KUKA KRL program: EPS_2_26115_SA6998_A_20260219035530.src

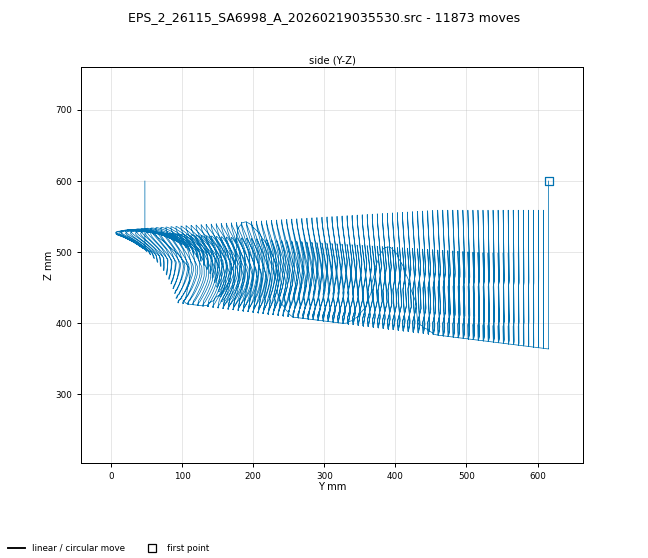
[picture p0: tool path of EPS_2_26115_SA6998_A_20260219035530.src, 11873 of 11875 moves have a stored position in this frame; points joined in program order, loops and branches not executed]
&ACCESS RVP
&REL 4
&COMMENT QRS 19112012
&PARAM EDITMASK = *
DEF PART()
EXT BAS (BAS_COMMAND :IN,REAL :IN )
INT I
BAS (#INITMOV,0 )

;KUKA QRS Post kuka4.cps  Date:22-06-2017 !

File_ID=3053

QRS_PRE_INIT()

;Init var - Until changes are made in qrs_pre_init
Outlet_Square_prg=0
Inlet_1_Square_prg=0
Inlet_2_Square_prg=0
Inlet_3_Square_prg=0
Inlet_4_Square_prg=0
Inlet_5_Square_prg=0

Outlet_1={X 0.000, Y 460.000, Z 458.500, B 0.000, E1 0.000 }
Inlet_1={X 0.000, Y 525.210, Z 398.500, B 0.000, E1 203.000 }
Outlet_1_type=201
Inlet_1_type=201
;QRS#1=Sidecore dimensions
;QRS#2=200-8" PVC SDR 35 Cut Back
;QRS#3=200-8" PVC SDR 35
;QRS#4=
;QRS#5=
;QRS#6=
;QRS#7=
;QRS#8=
;QRS#9=12-08 PSX
;QRS#10=12-08 PSX
;QRS#11=
;QRS#12=
;QRS#13=
;QRS#14=
;QRS#15=
;QRS#16=1220x127x838 2,75'
;QRS#17=EPS Height
;QRS#18=559
;QRS#19=*
;QRS#20= UPDATED VERSION 22-06-2017
;QRS#21=*
Outlet_Square=0100
Inlet_1_Square=0100
Inlet_2_Square=0
Inlet_3_Square=0
Inlet_4_Square=0
Inlet_5_Square=0
Mill_Square=1
Outlet_Square_Prg=214
Inlet_1_Square_prg=204

QRS_INIT()

$ADVANCE=5

; T1
PTP {E1 173.606,E2 173.606}
PTP {X 0,Y 615.505,A -85,B 0,C 180,E1 173.606,E2 173.606,E3 0,E4 0,E5 0,E6 0}
QRS_SPEED_INIT()
LIN {X 0,Y 615.505,Z 600,A -85,B 0,C 180,E1 173.606,E2 173.606,E3 0,E4 0,E5 0,E6 0} C_VEL
LIN {X 0,Y 615.505,Z 373.876,A -85,B 0,C 180,E1 173.606,E2 173.606} C_VEL
LIN {X 0,Y 615.505,Z 365.698,A -85,B 0,C 180,E1 173.606,E2 173.606} C_VEL
LIN {X 0,Y 615.491,Z 363.698,A -85,B 0,C 180,E1 173.42,E2 173.42} C_VEL
LIN {X 0,Y 615.494,Z 363.698,A -85,B 0,C 180,E1 170.801,E2 170.801} C_VEL
LIN {X 0,Y 615.477,Z 363.7,A -85,B 0,C 180,E1 168.139,E2 168.139} C_VEL
LIN {X 0,Y 615.491,Z 363.701,A -85,B 0,C 180,E1 165.451,E2 165.451} C_VEL
LIN {X 0,Y 615.482,Z 363.699,A -85,B 0,C 180,E1 162.729,E2 162.729} C_VEL
LIN {X 0,Y 615.481,Z 363.7,A -85,B 0,C 180,E1 159.967,E2 159.967} C_VEL
LIN {X 0,Y 615.493,Z 363.701,A -85,B 0,C 180,E1 157.156,E2 157.156} C_VEL
LIN {X 0,Y 615.477,Z 363.701,A -85,B 0,C 180,E1 154.284,E2 154.284} C_VEL
LIN {X 0,Y 615.487,Z 363.698,A -85,B 0,C 180,E1 151.55,E2 151.55} C_VEL
LIN {X 0,Y 615.492,Z 363.7,A -85,B 0,C 180,E1 148.914,E2 148.914} C_VEL
LIN {X 0,Y 615.48,Z 363.7,A -85,B 0,C 180,E1 146.467,E2 146.467} C_VEL
LIN {X 0,Y 615.492,Z 363.7,A -85,B 0,C 180,E1 143.575,E2 143.575} C_VEL
LIN {X 0,Y 615.482,Z 363.699,A -85,B 0,C 180,E1 140.939,E2 140.939} C_VEL
LIN {X 0,Y 615.491,Z 363.701,A -85,B 0,C 180,E1 138.526,E2 138.526} C_VEL
LIN {X 0,Y 615.48,Z 363.699,A -85,B 0,C 180,E1 135.85,E2 135.85} C_VEL
LIN {X 0,Y 615.482,Z 363.7,A -85,B 0,C 180,E1 133.047,E2 133.047} C_VEL
LIN {X 0,Y 615.472,Z 363.701,A -85,B 0,C 180,E1 130.608,E2 130.608} C_VEL
LIN {X 0,Y 615.489,Z 363.701,A -85,B 0,C 180,E1 128.012,E2 128.012} C_VEL
LIN {X 0,Y 615.498,Z 363.695,A -85,B 0,C 180,E1 125.616,E2 125.616} C_VEL
LIN {X 0,Y 615.489,Z 363.698,A -85,B 0,C 180,E1 123.237,E2 123.237} C_VEL
LIN {X 0,Y 615.496,Z 363.7,A -85,B 0,C 180,E1 120.92,E2 120.92} C_VEL
LIN {X 0,Y 615.478,Z 363.7,A -85,B 0,C 180,E1 118.448,E2 118.448} C_VEL
LIN {X 0,Y 615.486,Z 363.701,A -85,B 0,C 180,E1 115.568,E2 115.568} C_VEL
LIN {X 0,Y 615.48,Z 363.7,A -85,B 0,C 180,E1 112.846,E2 112.846} C_VEL
LIN {X 0,Y 615.489,Z 363.697,A -85,B 0,C 180,E1 110.034,E2 110.034} C_VEL
LIN {X 0,Y 615.491,Z 363.7,A -85,B 0,C 180,E1 107.271,E2 107.271} C_VEL
LIN {X 0,Y 615.481,Z 363.7,A -85,B 0,C 180,E1 104.55,E2 104.55} C_VEL
LIN {X 0,Y 615.478,Z 363.7,A -85,B 0,C 180,E1 102.531,E2 102.531} C_VEL
LIN {X 0,Y 615.489,Z 365.87,A -85,B 0,C 180,E1 100.528,E2 100.528} C_VEL
LIN {X 0,Y 615.493,Z 369.04,A -85,B 0,C 180,E1 97.877,E2 97.877} C_VEL
LIN {X 0,Y 615.456,Z 372.376,A -85,B 0,C 180,E1 95.243,E2 95.243} C_VEL
LIN {X 0,Y 615.448,Z 374.929,A -85,B 0,C 180,E1 93.274,E2 93.274} C_VEL
LIN {X 0,Y 615.441,Z 377.52,A -85,B 0,C 180,E1 91.31,E2 91.31} C_VEL
LIN {X 0,Y 615.434,Z 380.15,A -85,B 0,C 180,E1 89.347,E2 89.347} C_VEL
LIN {X 0,Y 615.428,Z 382.818,A -85,B 0,C 180,E1 87.383,E2 87.383} C_VEL
LIN {X 0,Y 615.426,Z 385.523,A -85,B 0,C 180,E1 85.416,E2 85.416} C_VEL
LIN {X 0,Y 615.431,Z 388.264,A -85,B 0,C 180,E1 83.444,E2 83.444} C_VEL
LIN {X 0,Y 615.434,Z 391.045,A -85,B 0,C 180,E1 81.464,E2 81.464} C_VEL
LIN {X 0,Y 615.435,Z 394.349,A -85,B 0,C 180,E1 79.138,E2 79.138} C_VEL
LIN {X 0,Y 615.478,Z 395.234,A -85,B 0,C 180,E1 78.537,E2 78.537} C_VEL
LIN {X 0,Y 615.495,Z 407.591,A -85,B 0,C 180,E1 78.266,E2 78.266} C_VEL
LIN {X 0,Y 615.465,Z 420.48,A -85,B 0,C 180,E1 77.848,E2 77.848} C_VEL
LIN {X 0,Y 615.439,Z 432.744,A -85,B 0,C 180,E1 77.303,E2 77.303} C_VEL
LIN {X 0,Y 615.477,Z 444.293,A -85,B 0,C 180,E1 76.632,E2 76.632} C_VEL
LIN {X 0,Y 615.498,Z 454.263,A -85,B 0,C 180,E1 75.911,E2 75.911} C_VEL
LIN {X 0,Y 615.497,Z 463.3,A -85,B 0,C 180,E1 75.115,E2 75.115} C_VEL
LIN {X 0,Y 615.496,Z 472.571,A -85,B 0,C 180,E1 74.097,E2 74.097} C_VEL
LIN {X 0,Y 615.497,Z 480.051,A -85,B 0,C 180,E1 73.074,E2 73.074} C_VEL
LIN {X 0,Y 615.497,Z 486.008,A -85,B 0,C 180,E1 72.045,E2 72.045} C_VEL
LIN {X 0,Y 615.496,Z 490.667,A -85,B 0,C 180,E1 71.01,E2 71.01} C_VEL
LIN {X 0,Y 615.498,Z 494.172,A -85,B 0,C 180,E1 69.969,E2 69.969} C_VEL
LIN {X 0,Y 615.492,Z 495.899,A -85,B 0,C 180,E1 69.271,E2 69.271} C_VEL
LIN {X 0,Y 615.497,Z 497.187,A -85,B 0,C 180,E1 68.57,E2 68.57} C_VEL
LIN {X 0,Y 615.491,Z 498.143,A -85,B 0,C 180,E1 67.654,E2 67.654} C_VEL
LIN {X 0,Y 615.496,Z 498.27,A -85,B 0,C 180,E1 66.446,E2 66.446} C_VEL
LIN {X 0,Y 615.494,Z 497.679,A -85,B 0,C 180,E1 65.73,E2 65.73} C_VEL
LIN {X 0,Y 615.495,Z 495.447,A -85,B 0,C 180,E1 64.43,E2 64.43} C_VEL
LIN {X 0,Y 615.498,Z 492.002,A -85,B 0,C 180,E1 63.257,E2 63.257} C_VEL
LIN {X 0,Y 615.495,Z 487.093,A -85,B 0,C 180,E1 62.087,E2 62.087} C_VEL
LIN {X 0,Y 615.496,Z 480.902,A -85,B 0,C 180,E1 60.971,E2 60.971} C_VEL
LIN {X 0,Y 615.497,Z 474.27,A -85,B 0,C 180,E1 60.023,E2 60.023} C_VEL
LIN {X 0,Y 615.497,Z 466.126,A -85,B 0,C 180,E1 59.083,E2 59.083} C_VEL
LIN {X 0,Y 615.499,Z 456.191,A -85,B 0,C 180,E1 58.156,E2 58.156} C_VEL
LIN {X 0,Y 615.496,Z 446.877,A -85,B 0,C 180,E1 57.448,E2 57.448} C_VEL
LIN {X 0,Y 615.477,Z 435.697,A -85,B 0,C 180,E1 56.765,E2 56.765} C_VEL
LIN {X 0,Y 615.487,Z 422.997,A -85,B 0,C 180,E1 56.163,E2 56.163} C_VEL
LIN {X 0,Y 615.486,Z 410.581,A -85,B 0,C 180,E1 55.726,E2 55.726} C_VEL
LIN {X 0,Y 615.492,Z 397.092,A -85,B 0,C 180,E1 55.407,E2 55.407} C_VEL
LIN {X 0,Y 615.489,Z 395.187,A -85,B 0,C 180,E1 55.364,E2 55.364} C_VEL
LIN {X 0,Y 615.474,Z 391.482,A -85,B 0,C 180,E1 52.759,E2 52.759} C_VEL
LIN {X 0,Y 615.493,Z 387.48,A -85,B 0,C 180,E1 49.911,E2 49.911} C_VEL
LIN {X 0,Y 615.479,Z 384.358,A -85,B 0,C 180,E1 47.649,E2 47.649} C_VEL
LIN {X 0,Y 615.46,Z 380.643,A -85,B 0,C 180,E1 44.932,E2 44.932} C_VEL
LIN {X 0,Y 615.495,Z 376.831,A -85,B 0,C 180,E1 42.084,E2 42.084} C_VEL
LIN {X 0,Y 615.45,Z 373.787,A -85,B 0,C 180,E1 39.753,E2 39.753} C_VEL
LIN {X 0,Y 615.457,Z 370.168,A -85,B 0,C 180,E1 36.936,E2 36.936} C_VEL
LIN {X 0,Y 615.495,Z 366.665,A -85,B 0,C 180,E1 34.022,E2 34.022} C_VEL
LIN {X 0,Y 615.485,Z 363.854,A -85,B 0,C 180,E1 31.686,E2 31.686} C_VEL
LIN {X 0,Y 615.463,Z 363.7,A -85,B 0,C 180,E1 29.408,E2 29.408} C_VEL
LIN {X 0,Y 615.481,Z 363.695,A -85,B 0,C 180,E1 27.049,E2 27.049} C_VEL
LIN {X 0,Y 615.471,Z 363.697,A -85,B 0,C 180,E1 24.273,E2 24.273} C_VEL
LIN {X 0,Y 615.486,Z 363.701,A -85,B 0,C 180,E1 22.137,E2 22.137} C_VEL
LIN {X 0,Y 615.491,Z 363.698,A -85,B 0,C 180,E1 19.338,E2 19.338} C_VEL
LIN {X 0,Y 615.466,Z 363.7,A -85,B 0,C 180,E1 16.432,E2 16.432} C_VEL
LIN {X 0,Y 615.478,Z 363.7,A -85,B 0,C 180,E1 13.874,E2 13.874} C_VEL
LIN {X 0,Y 615.489,Z 363.693,A -85,B 0,C 180,E1 10.902,E2 10.902} C_VEL
LIN {X 0,Y 615.482,Z 363.7,A -85,B 0,C 180,E1 8.537,E2 8.537} C_VEL
LIN {X 0,Y 615.49,Z 363.7,A -85,B 0,C 180,E1 5.898,E2 5.898} C_VEL
LIN {X 0,Y 615.49,Z 363.702,A -85,B 0,C 180,E1 3.273,E2 3.273} C_VEL
LIN {X 0,Y 615.491,Z 363.7,A -85,B 0,C 180,E1 0.654,E2 0.654} C_VEL
LIN {X 0,Y 615.486,Z 363.699,A -85,B 0,C 180,E1 -1.963,E2 -1.963} C_VEL
LIN {X 0,Y 615.476,Z 363.7,A -85,B 0,C 180,E1 -4.585,E2 -4.585} C_VEL
LIN {X 0,Y 615.492,Z 363.695,A -85,B 0,C 180,E1 -7.216,E2 -7.216} C_VEL
LIN {X 0,Y 615.468,Z 363.7,A -85,B 0,C 180,E1 -9.863,E2 -9.863} C_VEL
LIN {X 0,Y 615.468,Z 363.699,A -85,B 0,C 180,E1 -12.531,E2 -12.531} C_VEL
LIN {X 0,Y 615.483,Z 363.696,A -85,B 0,C 180,E1 -15.226,E2 -15.226} C_VEL
LIN {X 0,Y 615.465,Z 363.7,A -85,B 0,C 180,E1 -17.958,E2 -17.958} C_VEL
LIN {X 0,Y 615.493,Z 363.695,A -85,B 0,C 180,E1 -20.731,E2 -20.731} C_VEL
LIN {X 0,Y 615.486,Z 363.699,A -85,B 0,C 180,E1 -23.557,E2 -23.557} C_VEL
LIN {X 0,Y 615.458,Z 363.7,A -85,B 0,C 180,E1 -25.717,E2 -25.717} C_VEL
LIN {X 0,Y 615.481,Z 363.695,A -85,B 0,C 180,E1 -28.454,E2 -28.454} C_VEL
LIN {X 0,Y 615.469,Z 363.698,A -85,B 0,C 180,E1 -31.088,E2 -31.088} C_VEL
LIN {X 0,Y 615.468,Z 363.7,A -85,B 0,C 180,E1 -33.535,E2 -33.535} C_VEL
LIN {X 0,Y 615.491,Z 363.7,A -85,B 0,C 180,E1 -35.838,E2 -35.838} C_VEL
LIN {X 0,Y 615.463,Z 363.699,A -85,B 0,C 180,E1 -38.071,E2 -38.071} C_VEL
LIN {X 0,Y 615.492,Z 363.692,A -85,B 0,C 180,E1 -40.606,E2 -40.606} C_VEL
LIN {X 0,Y 615.459,Z 363.7,A -85,B 0,C 180,E1 -43.247,E2 -43.247} C_VEL
LIN {X 0,Y 615.472,Z 363.697,A -85,B 0,C 180,E1 -46.004,E2 -46.004} C_VEL
LIN {X 0,Y 615.475,Z 363.696,A -85,B 0,C 180,E1 -48.907,E2 -48.907} C_VEL
LIN {X 0,Y 615.47,Z 363.7,A -85,B 0,C 180,E1 -51.097,E2 -51.097} C_VEL
LIN {X 0,Y 615.483,Z 363.702,A -85,B 0,C 180,E1 -53.577,E2 -53.577} C_VEL
LIN {X 0,Y 615.493,Z 363.825,A -85,B 0,C 180,E1 -54.538,E2 -54.538} C_VEL
LIN {X 0,Y 615.444,Z 372.587,A -85,B 0,C 180,E1 -57.154,E2 -57.154} C_VEL
LIN {X 0,Y 615.423,Z 380.521,A -85,B 0,C 180,E1 -59.459,E2 -59.459} C_VEL
LIN {X 0,Y 615.479,Z 389.763,A -85,B 0,C 180,E1 -62.087,E2 -62.087} C_VEL
LIN {X 0,Y 615.455,Z 399.275,A -85,B 0,C 180,E1 -64.721,E2 -64.721} C_VEL
LIN {X 0,Y 615.46,Z 408.245,A -85,B 0,C 180,E1 -67.156,E2 -67.156} C_VEL
LIN {X 0,Y 615.489,Z 416.801,A -85,B 0,C 180,E1 -69.443,E2 -69.443} C_VEL
LIN {X 0,Y 615.486,Z 428.021,A -85,B 0,C 180,E1 -72.388,E2 -72.388} C_VEL
LIN {X 0,Y 615.482,Z 438.548,A -85,B 0,C 180,E1 -75.114,E2 -75.114} C_VEL
LIN {X 0,Y 615.469,Z 449.091,A -85,B 0,C 180,E1 -77.806,E2 -77.806} C_VEL
LIN {X 0,Y 615.494,Z 451.215,A -85,B 0,C 180,E1 -78.35,E2 -78.35} C_VEL
LIN {X 0,Y 615.497,Z 465.878,A -85,B 0,C 180,E1 -78.642,E2 -78.642} C_VEL
LIN {X 0,Y 615.457,Z 478.927,A -85,B 0,C 180,E1 -79.049,E2 -79.049} C_VEL
LIN {X 0,Y 615.452,Z 490.803,A -85,B 0,C 180,E1 -79.557,E2 -79.557} C_VEL
LIN {X 0,Y 615.496,Z 501.412,A -85,B 0,C 180,E1 -80.139,E2 -80.139} C_VEL
LIN {X 0,Y 615.498,Z 512.25,A -85,B 0,C 180,E1 -80.886,E2 -80.886} C_VEL
LIN {X 0,Y 615.497,Z 522.827,A -85,B 0,C 180,E1 -81.796,E2 -81.796} C_VEL
LIN {X 0,Y 615.497,Z 531.977,A -85,B 0,C 180,E1 -82.786,E2 -82.786} C_VEL
LIN {X 0,Y 615.497,Z 539.325,A -85,B 0,C 180,E1 -83.774,E2 -83.774} C_VEL
LIN {X 0,Y 615.498,Z 545.212,A -85,B 0,C 180,E1 -84.76,E2 -84.76} C_VEL
LIN {X 0,Y 615.494,Z 549.857,A -85,B 0,C 180,E1 -85.745,E2 -85.745} C_VEL
LIN {X 0,Y 615.494,Z 553.403,A -85,B 0,C 180,E1 -86.728,E2 -86.728} C_VEL
LIN {X 0,Y 615.497,Z 555.236,A -85,B 0,C 180,E1 -87.383,E2 -87.383} C_VEL
LIN {X 0,Y 615.499,Z 556.61,A -85,B 0,C 180,E1 -88.038,E2 -88.038} C_VEL
LIN {X 0,Y 615.496,Z 558.174,A -85,B 0,C 180,E1 -89.347,E2 -89.347} C_VEL
LIN {X 0,Y 615.494,Z 558.389,A -85,B 0,C 180,E1 -90.001,E2 -90.001} C_VEL
LIN {X 0,Y 615.495,Z 557.579,A -85,B 0,C 180,E1 -91.31,E2 -91.31} C_VEL
LIN {X 0,Y 615.499,Z 556.606,A -85,B 0,C 180,E1 -91.964,E2 -91.964} C_VEL
LIN {X 0,Y 615.497,Z 555.23,A -85,B 0,C 180,E1 -92.619,E2 -92.619} C_VEL
LIN {X 0,Y 615.496,Z 552.345,A -85,B 0,C 180,E1 -93.602,E2 -93.602} C_VEL
LIN {X 0,Y 615.498,Z 548.436,A -85,B 0,C 180,E1 -94.586,E2 -94.586} C_VEL
LIN {X 0,Y 615.499,Z 543.398,A -85,B 0,C 180,E1 -95.571,E2 -95.571} C_VEL
LIN {X 0,Y 615.497,Z 536.87,A -85,B 0,C 180,E1 -96.583,E2 -96.583} C_VEL
LIN {X 0,Y 615.497,Z 529.123,A -85,B 0,C 180,E1 -97.547,E2 -97.547} C_VEL
LIN {X 0,Y 615.498,Z 521.033,A -85,B 0,C 180,E1 -98.372,E2 -98.372} C_VEL
LIN {X 0,Y 615.499,Z 511.153,A -85,B 0,C 180,E1 -99.2,E2 -99.2} C_VEL
LIN {X 0,Y 615.487,Z 499.963,A -85,B 0,C 180,E1 -99.946,E2 -99.946} C_VEL
LIN {X 0,Y 615.449,Z 489.006,A -85,B 0,C 180,E1 -100.529,E2 -100.529} C_VEL
LIN {X 0,Y 615.463,Z 476.725,A -85,B 0,C 180,E1 -101.032,E2 -101.032} C_VEL
LIN {X 0,Y 615.499,Z 464.017,A -85,B 0,C 180,E1 -101.402,E2 -101.402} C_VEL
LIN {X 0,Y 615.495,Z 451.205,A -85,B 0,C 180,E1 -101.653,E2 -101.653} C_VEL
LIN {X 0,Y 615.471,Z 441.065,A -85,B 0,C 180,E1 -104.242,E2 -104.242} C_VEL
LIN {X 0,Y 615.49,Z 430.636,A -85,B 0,C 180,E1 -106.929,E2 -106.929} C_VEL
LIN {X 0,Y 615.484,Z 420.1,A -85,B 0,C 180,E1 -109.686,E2 -109.686} C_VEL
LIN {X 0,Y 615.491,Z 410.087,A -85,B 0,C 180,E1 -112.346,E2 -112.346} C_VEL
LIN {X 0,Y 615.445,Z 400.321,A -85,B 0,C 180,E1 -114.994,E2 -114.994} C_VEL
LIN {X 0,Y 615.476,Z 391.073,A -85,B 0,C 180,E1 -117.547,E2 -117.547} C_VEL
LIN {X 0,Y 615.439,Z 381.831,A -85,B 0,C 180,E1 -120.163,E2 -120.163} C_VEL
LIN {X 0,Y 615.433,Z 373.9,A -85,B 0,C 180,E1 -122.461,E2 -122.461} C_VEL
LIN {X 0,Y 615.46,Z 365.964,A -85,B 0,C 180,E1 -124.818,E2 -124.818} C_VEL
LIN {X 0,Y 615.495,Z 363.696,A -85,B 0,C 180,E1 -125.516,E2 -125.516} C_VEL
LIN {X 0,Y 615.491,Z 363.699,A -85,B 0,C 180,E1 -128.069,E2 -128.069} C_VEL
LIN {X 0,Y 615.481,Z 363.7,A -85,B 0,C 180,E1 -130.608,E2 -130.608} C_VEL
LIN {X 0,Y 615.484,Z 363.7,A -85,B 0,C 180,E1 -133.246,E2 -133.246} C_VEL
LIN {X 0,Y 615.473,Z 363.701,A -85,B 0,C 180,E1 -136.005,E2 -136.005} C_VEL
LIN {X 0,Y 615.491,Z 363.7,A -85,B 0,C 180,E1 -138.526,E2 -138.526} C_VEL
LIN {X 0,Y 615.484,Z 363.698,A -85,B 0,C 180,E1 -141.095,E2 -141.095} C_VEL
LIN {X 0,Y 615.494,Z 363.697,A -85,B 0,C 180,E1 -143.576,E2 -143.576} C_VEL
LIN {X 0,Y 615.492,Z 363.7,A -85,B 0,C 180,E1 -145.978,E2 -145.978} C_VEL
LIN {X 0,Y 615.477,Z 363.7,A -85,B 0,C 180,E1 -148.314,E2 -148.314} C_VEL
LIN {X 0,Y 615.475,Z 363.7,A -85,B 0,C 180,E1 -150.593,E2 -150.593} C_VEL
LIN {X 0,Y 615.486,Z 363.7,A -85,B 0,C 180,E1 -152.956,E2 -152.956} C_VEL
LIN {X 0,Y 615.476,Z 363.7,A -85,B 0,C 180,E1 -155.727,E2 -155.727} C_VEL
LIN {X 0,Y 615.474,Z 363.7,A -85,B 0,C 180,E1 -157.863,E2 -157.863} C_VEL
LIN {X 0,Y 615.486,Z 363.699,A -85,B 0,C 180,E1 -160.662,E2 -160.662} C_VEL
LIN {X 0,Y 615.488,Z 363.701,A -85,B 0,C 180,E1 -163.569,E2 -163.569} C_VEL
LIN {X 0,Y 615.473,Z 363.7,A -85,B 0,C 180,E1 -166.125,E2 -166.125} C_VEL
LIN {X 0,Y 615.495,Z 363.699,A -85,B 0,C 180,E1 -168.807,E2 -168.807} C_VEL
LIN {X 0,Y 615.488,Z 363.698,A -85,B 0,C 180,E1 -171.463,E2 -171.463} C_VEL
LIN {X 0,Y 615.482,Z 363.7,A -85,B 0,C 180,E1 -174.101,E2 -174.101} C_VEL
LIN {X 0,Y 615.482,Z 363.7,A -85,B 0,C 180,E1 -176.727,E2 -176.727} C_VEL
LIN {X 0,Y 615.479,Z 363.7,A -85,B 0,C 180,E1 -179.346,E2 -179.346} C_VEL
LIN {X 0,Y 615.485,Z 363.7,A -85,B 0,C 180,E1 -181.963,E2 -181.963} C_VEL
LIN {X 0,Y 615.488,Z 363.698,A -85,B 0,C 180,E1 -184.585,E2 -184.585} C_VEL
LIN {X 0,Y 615.491,Z 363.698,A -85,B 0,C 180,E1 -186.58,E2 -186.58} C_VEL
LIN {X 0,Y 614.818,Z 363.846,A -85,B 0,C 180,E1 -187.126,E2 -187.126} C_VEL
LIN {X 0,Y 611.987,Z 364.255,A -85,B 0,C 180,E1 -188.012,E2 -188.012} C_VEL
LIN {X 0,Y 609.594,Z 364.567,A -85,B 0,C 180,E1 -188.724,E2 -188.724} C_VEL
LIN {X 0,Y 608.554,Z 364.686,A -85,B 0,C 180,E1 -189.274,E2 -189.274} C_VEL
LIN {X 0,Y 608.461,Z 364.695,A -85,B 0,C 180,E1 -189.46,E2 -189.46} C_VEL
LIN {X 0,Y 608.457,Z 364.695,A -85,B 0,C 180,E1 -192,E2 -192} C_VEL
LIN {X 0,Y 608.478,Z 364.694,A -85,B 0,C 180,E1 -194.72,E2 -194.72} C_VEL
LIN {X 0,Y 608.449,Z 364.697,A -85,B 0,C 180,E1 -197.477,E2 -197.477} C_VEL
LIN {X 0,Y 608.459,Z 364.695,A -85,B 0,C 180,E1 -200.274,E2 -200.274} C_VEL
LIN {X 0,Y 608.452,Z 364.696,A -85,B 0,C 180,E1 -203.124,E2 -203.124} C_VEL
LIN {X 0,Y 608.464,Z 364.695,A -85,B 0,C 180,E1 -205.719,E2 -205.719} C_VEL
LIN {X 0,Y 608.451,Z 364.697,A -85,B 0,C 180,E1 -208.267,E2 -208.267} C_VEL
LIN {X 0,Y 608.479,Z 364.692,A -85,B 0,C 180,E1 -210.544,E2 -210.544} C_VEL
LIN {X 0,Y 608.463,Z 364.694,A -85,B 0,C 180,E1 -212.879,E2 -212.879} C_VEL
LIN {X 0,Y 608.441,Z 364.699,A -85,B 0,C 180,E1 -215.278,E2 -215.278} C_VEL
LIN {X 0,Y 608.464,Z 364.694,A -85,B 0,C 180,E1 -217.747,E2 -217.747} C_VEL
LIN {X 0,Y 608.448,Z 364.697,A -85,B 0,C 180,E1 -220.328,E2 -220.328} C_VEL
LIN {X 0,Y 608.467,Z 364.694,A -85,B 0,C 180,E1 -223.308,E2 -223.308} C_VEL
LIN {X 0,Y 608.472,Z 364.693,A -85,B 0,C 180,E1 -226.13,E2 -226.13} C_VEL
LIN {X 0,Y 608.456,Z 364.698,A -85,B 0,C 180,E1 -228.823,E2 -228.823} C_VEL
LIN {X 0,Y 608.441,Z 364.697,A -85,B 0,C 180,E1 -231.409,E2 -231.409} C_VEL
LIN {X 0,Y 608.453,Z 364.698,A -85,B 0,C 180,E1 -233.954,E2 -233.954} C_VEL
LIN {X 0,Y 608.47,Z 364.694,A -85,B 0,C 180,E1 -236.329,E2 -236.329} C_VEL
LIN {X 0,Y 608.466,Z 364.694,A -85,B 0,C 180,E1 -238.73,E2 -238.73} C_VEL
LIN {X 0,Y 608.473,Z 364.694,A -85,B 0,C 180,E1 -241.38,E2 -241.38} C_VEL
LIN {X 0,Y 608.479,Z 364.695,A -85,B 0,C 180,E1 -244.278,E2 -244.278} C_VEL
LIN {X 0,Y 608.45,Z 364.696,A -85,B 0,C 180,E1 -246.875,E2 -246.875} C_VEL
LIN {X 0,Y 608.47,Z 364.694,A -85,B 0,C 180,E1 -249.321,E2 -249.321} C_VEL
LIN {X 0,Y 608.453,Z 364.696,A -85,B 0,C 180,E1 -251.827,E2 -251.827} C_VEL
LIN {X 0,Y 608.474,Z 364.695,A -85,B 0,C 180,E1 -254.593,E2 -254.593} C_VEL
LIN {X 0,Y 608.473,Z 364.693,A -85,B 0,C 180,E1 -257.322,E2 -257.322} C_VEL
LIN {X 0,Y 608.428,Z 364.939,A -85,B 0,C 180,E1 -257.998,E2 -257.998} C_VEL
LIN {X 0,Y 608.435,Z 368.164,A -85,B 0,C 180,E1 -260.693,E2 -260.693} C_VEL
LIN {X 0,Y 608.418,Z 370.547,A -85,B 0,C 180,E1 -262.699,E2 -262.699} C_VEL
LIN {X 0,Y 608.392,Z 373.926,A -85,B 0,C 180,E1 -265.361,E2 -265.361} C_VEL
LIN {X 0,Y 608.464,Z 377.372,A -85,B 0,C 180,E1 -268.013,E2 -268.013} C_VEL
LIN {X 0,Y 608.382,Z 380.897,A -85,B 0,C 180,E1 -270.661,E2 -270.661} C_VEL
LIN {X 0,Y 608.362,Z 383.583,A -85,B 0,C 180,E1 -272.647,E2 -272.647} C_VEL
LIN {X 0,Y 608.362,Z 386.308,A -85,B 0,C 180,E1 -274.637,E2 -274.637} C_VEL
LIN {X 0,Y 608.385,Z 389.071,A -85,B 0,C 180,E1 -276.632,E2 -276.632} C_VEL
LIN {X 0,Y 608.38,Z 392.82,A -85,B 0,C 180,E1 -279.306,E2 -279.306} C_VEL
LIN {X 0,Y 608.407,Z 395.677,A -85,B 0,C 180,E1 -281.324,E2 -281.324} C_VEL
LIN {X 0,Y 608.544,Z 409.709,A -85,B 0,C 180,E1 -281.659,E2 -281.659} C_VEL
LIN {X 0,Y 608.495,Z 422.071,A -85,B 0,C 180,E1 -282.082,E2 -282.082} C_VEL
LIN {X 0,Y 608.459,Z 433.153,A -85,B 0,C 180,E1 -282.591,E2 -282.591} C_VEL
LIN {X 0,Y 608.475,Z 444.709,A -85,B 0,C 180,E1 -283.27,E2 -283.27} C_VEL
LIN {X 0,Y 608.472,Z 455.165,A -85,B 0,C 180,E1 -284.036,E2 -284.036} C_VEL
LIN {X 0,Y 608.468,Z 464.586,A -85,B 0,C 180,E1 -284.89,E2 -284.89} C_VEL
LIN {X 0,Y 608.461,Z 473.753,A -85,B 0,C 180,E1 -285.92,E2 -285.92} C_VEL
LIN {X 0,Y 608.46,Z 481.119,A -85,B 0,C 180,E1 -286.955,E2 -286.955} C_VEL
LIN {X 0,Y 608.455,Z 486.111,A -85,B 0,C 180,E1 -287.822,E2 -287.822} C_VEL
LIN {X 0,Y 608.456,Z 490.913,A -85,B 0,C 180,E1 -288.868,E2 -288.868} C_VEL
LIN {X 0,Y 608.436,Z 494.538,A -85,B 0,C 180,E1 -289.921,E2 -289.921} C_VEL
LIN {X 0,Y 608.423,Z 497.07,A -85,B 0,C 180,E1 -290.981,E2 -290.981} C_VEL
LIN {X 0,Y 608.417,Z 498.149,A -85,B 0,C 180,E1 -291.692,E2 -291.692} C_VEL
LIN {X 0,Y 608.423,Z 498.843,A -85,B 0,C 180,E1 -292.468,E2 -292.468} C_VEL
LIN {X 0,Y 608.432,Z 498.988,A -85,B 0,C 180,E1 -293.123,E2 -293.123} C_VEL
LIN {X 0,Y 608.422,Z 498.452,A -85,B 0,C 180,E1 -294.14,E2 -294.14} C_VEL
LIN {X 0,Y 608.439,Z 496.675,A -85,B 0,C 180,E1 -295.3,E2 -295.3} C_VEL
LIN {X 0,Y 608.432,Z 493.806,A -85,B 0,C 180,E1 -296.403,E2 -296.403} C_VEL
LIN {X 0,Y 608.436,Z 489.661,A -85,B 0,C 180,E1 -297.517,E2 -297.517} C_VEL
LIN {X 0,Y 608.433,Z 484.231,A -85,B 0,C 180,E1 -298.613,E2 -298.613} C_VEL
LIN {X 0,Y 608.46,Z 478.106,A -85,B 0,C 180,E1 -299.587,E2 -299.587} C_VEL
LIN {X 0,Y 608.455,Z 470.678,A -85,B 0,C 180,E1 -300.543,E2 -300.543} C_VEL
LIN {X 0,Y 608.478,Z 461.399,A -85,B 0,C 180,E1 -301.508,E2 -301.508} C_VEL
LIN {X 0,Y 608.497,Z 451.944,A -85,B 0,C 180,E1 -302.309,E2 -302.309} C_VEL
LIN {X 0,Y 608.498,Z 442.369,A -85,B 0,C 180,E1 -302.973,E2 -302.973} C_VEL
LIN {X 0,Y 608.515,Z 430.802,A -85,B 0,C 180,E1 -303.616,E2 -303.616} C_VEL
LIN {X 0,Y 608.531,Z 417.926,A -85,B 0,C 180,E1 -304.164,E2 -304.164} C_VEL
LIN {X 0,Y 608.558,Z 405.497,A -85,B 0,C 180,E1 -304.547,E2 -304.547} C_VEL
LIN {X 0,Y 608.426,Z 395.669,A -85,B 0,C 180,E1 -304.772,E2 -304.772} C_VEL
LIN {X 0,Y 608.415,Z 391.463,A -85,B 0,C 180,E1 -307.748,E2 -307.748} C_VEL
LIN {X 0,Y 608.419,Z 387.865,A -85,B 0,C 180,E1 -310.325,E2 -310.325} C_VEL
LIN {X 0,Y 608.403,Z 384.238,A -85,B 0,C 180,E1 -312.961,E2 -312.961} C_VEL
LIN {X 0,Y 608.439,Z 380.484,A -85,B 0,C 180,E1 -315.735,E2 -315.735} C_VEL
LIN {X 0,Y 608.433,Z 377.559,A -85,B 0,C 180,E1 -317.936,E2 -317.936} C_VEL
LIN {X 0,Y 608.382,Z 374.153,A -85,B 0,C 180,E1 -320.553,E2 -320.553} C_VEL
LIN {X 0,Y 608.401,Z 370.934,A -85,B 0,C 180,E1 -323.081,E2 -323.081} C_VEL
LIN {X 0,Y 608.453,Z 368.023,A -85,B 0,C 180,E1 -325.53,E2 -325.53} C_VEL
LIN {X 0,Y 608.425,Z 365.202,A -85,B 0,C 180,E1 -327.903,E2 -327.903} C_VEL
LIN {X 0,Y 608.463,Z 364.693,A -85,B 0,C 180,E1 -328.726,E2 -328.726} C_VEL
LIN {X 0,Y 608.446,Z 364.694,A -85,B 0,C 180,E1 -331.733,E2 -331.733} C_VEL
LIN {X 0,Y 608.445,Z 364.694,A -85,B 0,C 180,E1 -334.279,E2 -334.279} C_VEL
LIN {X 0,Y 608.452,Z 364.694,A -85,B 0,C 180,E1 -336.876,E2 -336.876} C_VEL
LIN {X 0,Y 608.445,Z 364.694,A -85,B 0,C 180,E1 -339.725,E2 -339.725} C_VEL
LIN {X 0,Y 608.444,Z 364.699,A -85,B 0,C 180,E1 -341.828,E2 -341.828} C_VEL
LIN {X 0,Y 608.465,Z 364.696,A -85,B 0,C 180,E1 -344.594,E2 -344.594} C_VEL
LIN {X 0,Y 608.463,Z 364.696,A -85,B 0,C 180,E1 -347.323,E2 -347.323} C_VEL
LIN {X 0,Y 608.451,Z 364.697,A -85,B 0,C 180,E1 -350.023,E2 -350.023} C_VEL
LIN {X 0,Y 608.478,Z 364.695,A -85,B 0,C 180,E1 -352.701,E2 -352.701} C_VEL
LIN {X 0,Y 608.456,Z 364.698,A -85,B 0,C 180,E1 -355.362,E2 -355.362} C_VEL
LIN {X 0,Y 608.467,Z 364.696,A -85,B 0,C 180,E1 -358.014,E2 -358.014} C_VEL
LIN {X 0,Y 608.479,Z 364.694,A -85,B 0,C 180,E1 -360.662,E2 -360.662} C_VEL
LIN {X 0,Y 608.483,Z 364.693,A -85,B 0,C 180,E1 -363.311,E2 -363.311} C_VEL
LIN {X 0,Y 608.448,Z 364.696,A -85,B 0,C 180,E1 -365.967,E2 -365.967} C_VEL
LIN {X 0,Y 608.439,Z 364.697,A -85,B 0,C 180,E1 -368.636,E2 -368.636} C_VEL
LIN {X 0,Y 608.469,Z 364.693,A -85,B 0,C 180,E1 -371.324,E2 -371.324} C_VEL
LIN {X 0,Y 608.447,Z 364.696,A -85,B 0,C 180,E1 -374.038,E2 -374.038} C_VEL
LIN {X 0,Y 608.462,Z 364.695,A -85,B 0,C 180,E1 -376.784,E2 -376.784} C_VEL
LIN {X 0,Y 608.444,Z 364.698,A -85,B 0,C 180,E1 -379.571,E2 -379.571} C_VEL
LIN {X 0,Y 608.475,Z 364.694,A -85,B 0,C 180,E1 -382.486,E2 -382.486} C_VEL
LIN {X 0,Y 608.442,Z 364.697,A -85,B 0,C 180,E1 -385.302,E2 -385.302} C_VEL
LIN {X 0,Y 608.44,Z 364.697,A -85,B 0,C 180,E1 -387.519,E2 -387.519} C_VEL
LIN {X 0,Y 608.443,Z 364.695,A -85,B 0,C 180,E1 -389.972,E2 -389.972} C_VEL
LIN {X 0,Y 608.461,Z 364.692,A -85,B 0,C 180,E1 -392.526,E2 -392.526} C_VEL
LIN {X 0,Y 608.43,Z 364.696,A -85,B 0,C 180,E1 -395.279,E2 -395.279} C_VEL
LIN {X 0,Y 608.454,Z 364.694,A -85,B 0,C 180,E1 -397.748,E2 -397.748} C_VEL
LIN {X 0,Y 608.467,Z 364.693,A -85,B 0,C 180,E1 -400.334,E2 -400.334} C_VEL
LIN {X 0,Y 608.449,Z 364.694,A -85,B 0,C 180,E1 -403.31,E2 -403.31} C_VEL
LIN {X 0,Y 608.46,Z 364.693,A -85,B 0,C 180,E1 -406.133,E2 -406.133} C_VEL
LIN {X 0,Y 608.448,Z 364.694,A -85,B 0,C 180,E1 -408.826,E2 -408.826} C_VEL
LIN {X 0,Y 608.456,Z 364.693,A -85,B 0,C 180,E1 -411.414,E2 -411.414} C_VEL
LIN {X 0,Y 608.487,Z 364.699,A -85,B 0,C 180,E1 -414.334,E2 -414.334} C_VEL
LIN {X 0,Y 608.519,Z 372.6,A -85,B 0,C 180,E1 -416.732,E2 -416.732} C_VEL
LIN {X 0,Y 608.467,Z 380.604,A -85,B 0,C 180,E1 -419.09,E2 -419.09} C_VEL
LIN {X 0,Y 608.451,Z 389.811,A -85,B 0,C 180,E1 -421.735,E2 -421.735} C_VEL
LIN {X 0,Y 608.516,Z 398.839,A -85,B 0,C 180,E1 -424.271,E2 -424.271} C_VEL
LIN {X 0,Y 608.438,Z 408.345,A -85,B 0,C 180,E1 -426.877,E2 -426.877} C_VEL
LIN {X 0,Y 608.466,Z 417.417,A -85,B 0,C 180,E1 -429.323,E2 -429.323} C_VEL
LIN {X 0,Y 608.448,Z 428.203,A -85,B 0,C 180,E1 -432.178,E2 -432.178} C_VEL
LIN {X 0,Y 608.438,Z 438.794,A -85,B 0,C 180,E1 -434.938,E2 -434.938} C_VEL
LIN {X 0,Y 608.406,Z 448.061,A -85,B 0,C 180,E1 -437.323,E2 -437.323} C_VEL
LIN {X 0,Y 608.441,Z 451.578,A -85,B 0,C 180,E1 -438.223,E2 -438.223} C_VEL
LIN {X 0,Y 608.547,Z 465.16,A -85,B 0,C 180,E1 -438.489,E2 -438.489} C_VEL
LIN {X 0,Y 608.488,Z 478.508,A -85,B 0,C 180,E1 -438.902,E2 -438.902} C_VEL
LIN {X 0,Y 608.478,Z 490.952,A -85,B 0,C 180,E1 -439.436,E2 -439.436} C_VEL
LIN {X 0,Y 608.486,Z 501.603,A -85,B 0,C 180,E1 -440.025,E2 -440.025} C_VEL
LIN {X 0,Y 608.483,Z 512.493,A -85,B 0,C 180,E1 -440.78,E2 -440.78} C_VEL
LIN {X 0,Y 608.474,Z 523.127,A -85,B 0,C 180,E1 -441.7,E2 -441.7} C_VEL
LIN {X 0,Y 608.47,Z 530.973,A -85,B 0,C 180,E1 -442.535,E2 -442.535} C_VEL
LIN {X 0,Y 608.46,Z 538.292,A -85,B 0,C 180,E1 -443.485,E2 -443.485} C_VEL
LIN {X 0,Y 608.45,Z 543.874,A -85,B 0,C 180,E1 -444.367,E2 -444.367} C_VEL
LIN {X 0,Y 608.432,Z 548.956,A -85,B 0,C 180,E1 -445.364,E2 -445.364} C_VEL
LIN {X 0,Y 608.449,Z 552.901,A -85,B 0,C 180,E1 -446.359,E2 -446.359} C_VEL
LIN {X 0,Y 608.425,Z 555.812,A -85,B 0,C 180,E1 -447.353,E2 -447.353} C_VEL
LIN {X 0,Y 608.444,Z 557.203,A -85,B 0,C 180,E1 -448.015,E2 -448.015} C_VEL
LIN {X 0,Y 608.438,Z 558.784,A -85,B 0,C 180,E1 -449.339,E2 -449.339} C_VEL
LIN {X 0,Y 608.434,Z 559,A -85,B 0,C 180,E1 -450.001,E2 -450.001} C_VEL
LIN {X 0,Y 608.448,Z 558.182,A -85,B 0,C 180,E1 -451.325,E2 -451.325} C_VEL
LIN {X 0,Y 608.444,Z 557.199,A -85,B 0,C 180,E1 -451.987,E2 -451.987} C_VEL
LIN {X 0,Y 608.425,Z 555.806,A -85,B 0,C 180,E1 -452.649,E2 -452.649} C_VEL
LIN {X 0,Y 608.449,Z 552.892,A -85,B 0,C 180,E1 -453.644,E2 -453.644} C_VEL
LIN {X 0,Y 608.432,Z 548.945,A -85,B 0,C 180,E1 -454.639,E2 -454.639} C_VEL
LIN {X 0,Y 608.437,Z 542.869,A -85,B 0,C 180,E1 -455.802,E2 -455.802} C_VEL
LIN {X 0,Y 608.463,Z 536.226,A -85,B 0,C 180,E1 -456.8,E2 -456.8} C_VEL
LIN {X 0,Y 608.456,Z 527.979,A -85,B 0,C 180,E1 -457.801,E2 -457.801} C_VEL
LIN {X 0,Y 608.472,Z 519.523,A -85,B 0,C 180,E1 -458.637,E2 -458.637} C_VEL
LIN {X 0,Y 608.481,Z 509.075,A -85,B 0,C 180,E1 -459.474,E2 -459.474} C_VEL
LIN {X 0,Y 608.499,Z 498.737,A -85,B 0,C 180,E1 -460.146,E2 -460.146} C_VEL
LIN {X 0,Y 608.472,Z 487.813,A -85,B 0,C 180,E1 -460.715,E2 -460.715} C_VEL
LIN {X 0,Y 608.495,Z 476.04,A -85,B 0,C 180,E1 -461.188,E2 -461.188} C_VEL
LIN {X 0,Y 608.55,Z 463.221,A -85,B 0,C 180,E1 -461.555,E2 -461.555} C_VEL
LIN {X 0,Y 608.444,Z 451.526,A -85,B 0,C 180,E1 -461.79,E2 -461.79} C_VEL
LIN {X 0,Y 608.435,Z 441.432,A -85,B 0,C 180,E1 -464.381,E2 -464.381} C_VEL
LIN {X 0,Y 608.445,Z 430.841,A -85,B 0,C 180,E1 -467.131,E2 -467.131} C_VEL
LIN {X 0,Y 608.455,Z 421.573,A -85,B 0,C 180,E1 -469.571,E2 -469.571} C_VEL
LIN {X 0,Y 608.465,Z 410.722,A -85,B 0,C 180,E1 -472.477,E2 -472.477} C_VEL
LIN {X 0,Y 608.435,Z 401.715,A -85,B 0,C 180,E1 -474.937,E2 -474.937} C_VEL
LIN {X 0,Y 608.446,Z 393.579,A -85,B 0,C 180,E1 -477.201,E2 -477.201} C_VEL
LIN {X 0,Y 608.476,Z 383.837,A -85,B 0,C 180,E1 -479.972,E2 -479.972} C_VEL
LIN {X 0,Y 608.482,Z 375.105,A -85,B 0,C 180,E1 -482.525,E2 -482.525} C_VEL
LIN {X 0,Y 608.557,Z 365.971,A -85,B 0,C 180,E1 -485.271,E2 -485.271} C_VEL
LIN {X 0,Y 608.487,Z 364.692,A -85,B 0,C 180,E1 -485.682,E2 -485.682} C_VEL
LIN {X 0,Y 608.47,Z 364.696,A -85,B 0,C 180,E1 -488.24,E2 -488.24} C_VEL
LIN {X 0,Y 608.466,Z 364.696,A -85,B 0,C 180,E1 -491.342,E2 -491.342} C_VEL
LIN {X 0,Y 608.45,Z 364.697,A -85,B 0,C 180,E1 -494.263,E2 -494.263} C_VEL
LIN {X 0,Y 608.449,Z 364.696,A -85,B 0,C 180,E1 -497.04,E2 -497.04} C_VEL
LIN {X 0,Y 608.457,Z 364.697,A -85,B 0,C 180,E1 -499.697,E2 -499.697} C_VEL
LIN {X 0,Y 608.483,Z 364.694,A -85,B 0,C 180,E1 -502.841,E2 -502.841} C_VEL
LIN {X 0,Y 608.477,Z 364.693,A -85,B 0,C 180,E1 -505.531,E2 -505.531} C_VEL
LIN {X 0,Y 608.468,Z 364.696,A -85,B 0,C 180,E1 -507.906,E2 -507.906} C_VEL
LIN {X 0,Y 608.471,Z 364.694,A -85,B 0,C 180,E1 -510.22,E2 -510.22} C_VEL
LIN {X 0,Y 608.476,Z 364.693,A -85,B 0,C 180,E1 -512.794,E2 -512.794} C_VEL
LIN {X 0,Y 608.448,Z 364.697,A -85,B 0,C 180,E1 -515.429,E2 -515.429} C_VEL
LIN {X 0,Y 608.464,Z 364.697,A -85,B 0,C 180,E1 -518.308,E2 -518.308} C_VEL
LIN {X 0,Y 608.479,Z 364.694,A -85,B 0,C 180,E1 -521.282,E2 -521.282} C_VEL
LIN {X 0,Y 608.455,Z 364.695,A -85,B 0,C 180,E1 -523.906,E2 -523.906} C_VEL
LIN {X 0,Y 608.466,Z 364.696,A -85,B 0,C 180,E1 -526.644,E2 -526.644} C_VEL
LIN {X 0,Y 608.47,Z 364.693,A -85,B 0,C 180,E1 -529.35,E2 -529.35} C_VEL
LIN {X 0,Y 608.473,Z 364.694,A -85,B 0,C 180,E1 -532.033,E2 -532.033} C_VEL
LIN {X 0,Y 608.466,Z 364.695,A -85,B 0,C 180,E1 -534.698,E2 -534.698} C_VEL
LIN {X 0,Y 608.47,Z 364.693,A -85,B 0,C 180,E1 -537.352,E2 -537.352} C_VEL
LIN {X 0,Y 608.478,Z 364.694,A -85,B 0,C 180,E1 -540,E2 -540} C_VEL
LIN {X 0,Y 608.477,Z 364.692,A -85,B 0,C 180,E1 -542.648,E2 -542.648} C_VEL
LIN {X 0,Y 608.474,Z 364.695,A -85,B 0,C 180,E1 -545.302,E2 -545.302} C_VEL
LIN {X 0,Y 608.471,Z 364.693,A -85,B 0,C 180,E1 -547.967,E2 -547.967} C_VEL
LIN {X 0,Y 608.461,Z 364.695,A -85,B 0,C 180,E1 -549.46,E2 -549.46} C_VEL
LIN {X 0,Y 607.775,Z 364.78,A -85,B 0,C 180,E1 -550.013,E2 -550.013} C_VEL
LIN {X 0,Y 604.917,Z 365.136,A -85,B 0,C 180,E1 -550.91,E2 -550.91} C_VEL
LIN {X 0,Y 602.518,Z 365.436,A -85,B 0,C 180,E1 -551.631,E2 -551.631} C_VEL
LIN {X 0,Y 601.492,Z 365.563,A -85,B 0,C 180,E1 -552.188,E2 -552.188} C_VEL
LIN {X 0,Y 601.41,Z 365.572,A -85,B 0,C 180,E1 -552.376,E2 -552.376} C_VEL
LIN {X 0,Y 601.432,Z 365.57,A -85,B 0,C 180,E1 -554.897,E2 -554.897} C_VEL
LIN {X 0,Y 601.434,Z 365.57,A -85,B 0,C 180,E1 -556.986,E2 -556.986} C_VEL
LIN {X 0,Y 601.402,Z 365.576,A -85,B 0,C 180,E1 -559.81,E2 -559.81} C_VEL
LIN {X 0,Y 601.419,Z 365.572,A -85,B 0,C 180,E1 -562.605,E2 -562.605} C_VEL
LIN {X 0,Y 601.402,Z 365.576,A -85,B 0,C 180,E1 -564.879,E2 -564.879} C_VEL
LIN {X 0,Y 601.419,Z 365.572,A -85,B 0,C 180,E1 -567.362,E2 -567.362} C_VEL
LIN {X 0,Y 601.432,Z 365.572,A -85,B 0,C 180,E1 -570.164,E2 -570.164} C_VEL
LIN {X 0,Y 601.429,Z 365.57,A -85,B 0,C 180,E1 -572.716,E2 -572.716} C_VEL
LIN {X 0,Y 601.399,Z 365.575,A -85,B 0,C 180,E1 -575.112,E2 -575.112} C_VEL
LIN {X 0,Y 601.437,Z 365.572,A -85,B 0,C 180,E1 -577.419,E2 -577.419} C_VEL
LIN {X 0,Y 601.404,Z 365.573,A -85,B 0,C 180,E1 -579.996,E2 -579.996} C_VEL
LIN {X 0,Y 601.41,Z 365.575,A -85,B 0,C 180,E1 -582.671,E2 -582.671} C_VEL
LIN {X 0,Y 601.402,Z 365.575,A -85,B 0,C 180,E1 -585.479,E2 -585.479} C_VEL
LIN {X 0,Y 601.43,Z 365.57,A -85,B 0,C 180,E1 -588.406,E2 -588.406} C_VEL
LIN {X 0,Y 601.435,Z 365.572,A -85,B 0,C 180,E1 -590.875,E2 -590.875} C_VEL
LIN {X 0,Y 601.407,Z 365.573,A -85,B 0,C 180,E1 -593.417,E2 -593.417} C_VEL
LIN {X 0,Y 601.437,Z 365.572,A -85,B 0,C 180,E1 -596.064,E2 -596.064} C_VEL
LIN {X 0,Y 601.418,Z 365.574,A -85,B 0,C 180,E1 -599.057,E2 -599.057} C_VEL
LIN {X 0,Y 601.433,Z 365.571,A -85,B 0,C 180,E1 -601.372,E2 -601.372} C_VEL
LIN {X 0,Y 601.418,Z 365.573,A -85,B 0,C 180,E1 -604.132,E2 -604.132} C_VEL
LIN {X 0,Y 601.421,Z 365.573,A -85,B 0,C 180,E1 -606.589,E2 -606.589} C_VEL
LIN {X 0,Y 601.435,Z 365.572,A -85,B 0,C 180,E1 -609.477,E2 -609.477} C_VEL
LIN {X 0,Y 601.403,Z 365.574,A -85,B 0,C 180,E1 -612.311,E2 -612.311} C_VEL
LIN {X 0,Y 601.418,Z 365.572,A -85,B 0,C 180,E1 -614.408,E2 -614.408} C_VEL
LIN {X 0,Y 601.421,Z 365.571,A -85,B 0,C 180,E1 -617.171,E2 -617.171} C_VEL
LIN {X 0,Y 601.378,Z 365.579,A -85,B 0,C 180,E1 -617.856,E2 -617.856} C_VEL
LIN {X 0,Y 601.402,Z 367.817,A -85,B 0,C 180,E1 -619.903,E2 -619.903} C_VEL
LIN {X 0,Y 601.354,Z 371.016,A -85,B 0,C 180,E1 -622.613,E2 -622.613} C_VEL
LIN {X 0,Y 601.332,Z 374.305,A -85,B 0,C 180,E1 -625.306,E2 -625.306} C_VEL
LIN {X 0,Y 601.372,Z 377.752,A -85,B 0,C 180,E1 -627.99,E2 -627.99} C_VEL
LIN {X 0,Y 601.31,Z 381.275,A -85,B 0,C 180,E1 -630.668,E2 -630.668} C_VEL
LIN {X 0,Y 601.269,Z 383.963,A -85,B 0,C 180,E1 -632.678,E2 -632.678} C_VEL
LIN {X 0,Y 601.297,Z 387.605,A -85,B 0,C 180,E1 -635.364,E2 -635.364} C_VEL
LIN {X 0,Y 601.314,Z 391.319,A -85,B 0,C 180,E1 -638.061,E2 -638.061} C_VEL
LIN {X 0,Y 601.287,Z 395.341,A -85,B 0,C 180,E1 -640.943,E2 -640.943} C_VEL
LIN {X 0,Y 601.3,Z 395.672,A -85,B 0,C 180,E1 -641.179,E2 -641.179} C_VEL
LIN {X 0,Y 601.585,Z 401.505,A -85,B 0,C 180,E1 -641.314,E2 -641.314} C_VEL
LIN {X 0,Y 601.579,Z 414.234,A -85,B 0,C 180,E1 -641.667,E2 -641.667} C_VEL
LIN {X 0,Y 601.475,Z 426.408,A -85,B 0,C 180,E1 -642.14,E2 -642.14} C_VEL
LIN {X 0,Y 601.456,Z 438.085,A -85,B 0,C 180,E1 -642.74,E2 -642.74} C_VEL
LIN {X 0,Y 601.455,Z 448.646,A -85,B 0,C 180,E1 -643.427,E2 -643.427} C_VEL
LIN {X 0,Y 601.43,Z 458.35,A -85,B 0,C 180,E1 -644.204,E2 -644.204} C_VEL
LIN {X 0,Y 601.388,Z 467.24,A -85,B 0,C 180,E1 -645.07,E2 -645.07} C_VEL
LIN {X 0,Y 601.404,Z 475.842,A -85,B 0,C 180,E1 -646.112,E2 -646.112} C_VEL
LIN {X 0,Y 601.389,Z 482.784,A -85,B 0,C 180,E1 -647.161,E2 -647.161} C_VEL
LIN {X 0,Y 601.358,Z 487.476,A -85,B 0,C 180,E1 -648.04,E2 -648.04} C_VEL
LIN {X 0,Y 601.343,Z 491.955,A -85,B 0,C 180,E1 -649.1,E2 -649.1} C_VEL
LIN {X 0,Y 601.332,Z 494.32,A -85,B 0,C 180,E1 -649.81,E2 -649.81} C_VEL
LIN {X 0,Y 601.338,Z 496.698,A -85,B 0,C 180,E1 -650.775,E2 -650.775} C_VEL
LIN {X 0,Y 601.335,Z 498.479,A -85,B 0,C 180,E1 -651.96,E2 -651.96} C_VEL
LIN {X 0,Y 601.318,Z 498.923,A -85,B 0,C 180,E1 -652.685,E2 -652.685} C_VEL
LIN {X 0,Y 601.325,Z 498.921,A -85,B 0,C 180,E1 -653.412,E2 -653.412} C_VEL
LIN {X 0,Y 601.318,Z 498.32,A -85,B 0,C 180,E1 -654.267,E2 -654.267} C_VEL
LIN {X 0,Y 601.33,Z 497.488,A -85,B 0,C 180,E1 -654.88,E2 -654.88} C_VEL
LIN {X 0,Y 601.337,Z 495.474,A -85,B 0,C 180,E1 -655.852,E2 -655.852} C_VEL
LIN {X 0,Y 601.333,Z 491.497,A -85,B 0,C 180,E1 -657.115,E2 -657.115} C_VEL
LIN {X 0,Y 601.374,Z 486.531,A -85,B 0,C 180,E1 -658.247,E2 -658.247} C_VEL
LIN {X 0,Y 601.376,Z 479.911,A -85,B 0,C 180,E1 -659.393,E2 -659.393} C_VEL
LIN {X 0,Y 601.4,Z 472.923,A -85,B 0,C 180,E1 -660.357,E2 -660.357} C_VEL
LIN {X 0,Y 601.413,Z 464.765,A -85,B 0,C 180,E1 -661.278,E2 -661.278} C_VEL
LIN {X 0,Y 601.44,Z 455.702,A -85,B 0,C 180,E1 -662.117,E2 -662.117} C_VEL
LIN {X 0,Y 601.48,Z 445.323,A -85,B 0,C 180,E1 -662.894,E2 -662.894} C_VEL
LIN {X 0,Y 601.494,Z 433.404,A -85,B 0,C 180,E1 -663.608,E2 -663.608} C_VEL
LIN {X 0,Y 601.542,Z 421.495,A -85,B 0,C 180,E1 -664.159,E2 -664.159} C_VEL
LIN {X 0,Y 601.566,Z 408.433,A -85,B 0,C 180,E1 -664.601,E2 -664.601} C_VEL
LIN {X 0,Y 601.411,Z 396.583,A -85,B 0,C 180,E1 -664.879,E2 -664.879} C_VEL
LIN {X 0,Y 601.337,Z 395.673,A -85,B 0,C 180,E1 -664.909,E2 -664.909} C_VEL
LIN {X 0,Y 601.316,Z 392.157,A -85,B 0,C 180,E1 -667.425,E2 -667.425} C_VEL
LIN {X 0,Y 601.331,Z 388.6,A -85,B 0,C 180,E1 -669.999,E2 -669.999} C_VEL
LIN {X 0,Y 601.322,Z 384.954,A -85,B 0,C 180,E1 -672.675,E2 -672.675} C_VEL
LIN {X 0,Y 601.348,Z 381.203,A -85,B 0,C 180,E1 -675.475,E2 -675.475} C_VEL
LIN {X 0,Y 601.314,Z 377.593,A -85,B 0,C 180,E1 -678.225,E2 -678.225} C_VEL
LIN {X 0,Y 601.296,Z 374.205,A -85,B 0,C 180,E1 -680.864,E2 -680.864} C_VEL
LIN {X 0,Y 601.344,Z 370.788,A -85,B 0,C 180,E1 -683.743,E2 -683.743} C_VEL
LIN {X 0,Y 601.375,Z 368.046,A -85,B 0,C 180,E1 -686.069,E2 -686.069} C_VEL
LIN {X 0,Y 601.362,Z 365.582,A -85,B 0,C 180,E1 -688.271,E2 -688.271} C_VEL
LIN {X 0,Y 601.402,Z 365.572,A -85,B 0,C 180,E1 -690.606,E2 -690.606} C_VEL
LIN {X 0,Y 601.444,Z 365.567,A -85,B 0,C 180,E1 -692.889,E2 -692.889} C_VEL
LIN {X 0,Y 601.441,Z 365.567,A -85,B 0,C 180,E1 -695.859,E2 -695.859} C_VEL
LIN {X 0,Y 601.404,Z 365.573,A -85,B 0,C 180,E1 -698.04,E2 -698.04} C_VEL
LIN {X 0,Y 601.419,Z 365.57,A -85,B 0,C 180,E1 -700.901,E2 -700.901} C_VEL
LIN {X 0,Y 601.418,Z 365.57,A -85,B 0,C 180,E1 -703.713,E2 -703.713} C_VEL
LIN {X 0,Y 601.402,Z 365.571,A -85,B 0,C 180,E1 -706.484,E2 -706.484} C_VEL
LIN {X 0,Y 601.416,Z 365.57,A -85,B 0,C 180,E1 -709.224,E2 -709.224} C_VEL
LIN {X 0,Y 601.42,Z 365.569,A -85,B 0,C 180,E1 -711.939,E2 -711.939} C_VEL
LIN {X 0,Y 601.424,Z 365.569,A -85,B 0,C 180,E1 -714.636,E2 -714.636} C_VEL
LIN {X 0,Y 601.433,Z 365.568,A -85,B 0,C 180,E1 -717.321,E2 -717.321} C_VEL
LIN {X 0,Y 601.418,Z 365.57,A -85,B 0,C 180,E1 -720,E2 -720} C_VEL
LIN {X 0,Y 601.438,Z 365.567,A -85,B 0,C 180,E1 -722.679,E2 -722.679} C_VEL
LIN {X 0,Y 601.415,Z 365.57,A -85,B 0,C 180,E1 -725.364,E2 -725.364} C_VEL
LIN {X 0,Y 601.421,Z 365.569,A -85,B 0,C 180,E1 -728.061,E2 -728.061} C_VEL
LIN {X 0,Y 601.42,Z 365.569,A -85,B 0,C 180,E1 -731.022,E2 -731.022} C_VEL
LIN {X 0,Y 601.4,Z 365.572,A -85,B 0,C 180,E1 -733.516,E2 -733.516} C_VEL
LIN {X 0,Y 601.425,Z 365.569,A -85,B 0,C 180,E1 -736.287,E2 -736.287} C_VEL
LIN {X 0,Y 601.419,Z 365.569,A -85,B 0,C 180,E1 -739.099,E2 -739.099} C_VEL
LIN {X 0,Y 601.403,Z 365.572,A -85,B 0,C 180,E1 -741.96,E2 -741.96} C_VEL
LIN {X 0,Y 601.427,Z 365.569,A -85,B 0,C 180,E1 -744.296,E2 -744.296} C_VEL
LIN {X 0,Y 601.439,Z 365.567,A -85,B 0,C 180,E1 -747.112,E2 -747.112} C_VEL
LIN {X 0,Y 601.403,Z 365.574,A -85,B 0,C 180,E1 -749.394,E2 -749.394} C_VEL
LIN {X 0,Y 601.405,Z 365.575,A -85,B 0,C 180,E1 -751.727,E2 -751.727} C_VEL
LIN {X 0,Y 601.415,Z 365.571,A -85,B 0,C 180,E1 -754.119,E2 -754.119} C_VEL
LIN {X 0,Y 601.409,Z 365.571,A -85,B 0,C 180,E1 -756.583,E2 -756.583} C_VEL
LIN {X 0,Y 601.402,Z 365.572,A -85,B 0,C 180,E1 -759.535,E2 -759.535} C_VEL
LIN {X 0,Y 601.412,Z 365.571,A -85,B 0,C 180,E1 -761.766,E2 -761.766} C_VEL
LIN {X 0,Y 601.411,Z 365.571,A -85,B 0,C 180,E1 -764.537,E2 -764.537} C_VEL
LIN {X 0,Y 601.396,Z 365.573,A -85,B 0,C 180,E1 -767.331,E2 -767.331} C_VEL
LIN {X 0,Y 601.405,Z 365.571,A -85,B 0,C 180,E1 -770.007,E2 -770.007} C_VEL
LIN {X 0,Y 601.426,Z 365.57,A -85,B 0,C 180,E1 -772.619,E2 -772.619} C_VEL
LIN {X 0,Y 601.468,Z 365.692,A -85,B 0,C 180,E1 -774.163,E2 -774.163} C_VEL
LIN {X 0,Y 601.583,Z 372.851,A -85,B 0,C 180,E1 -776.373,E2 -776.373} C_VEL
LIN {X 0,Y 601.497,Z 381.867,A -85,B 0,C 180,E1 -779.065,E2 -779.065} C_VEL
LIN {X 0,Y 601.451,Z 389.811,A -85,B 0,C 180,E1 -781.376,E2 -781.376} C_VEL
LIN {X 0,Y 601.491,Z 399.442,A -85,B 0,C 180,E1 -784.118,E2 -784.118} C_VEL
LIN {X 0,Y 601.41,Z 409.669,A -85,B 0,C 180,E1 -786.956,E2 -786.956} C_VEL
LIN {X 0,Y 601.431,Z 418.936,A -85,B 0,C 180,E1 -789.48,E2 -789.48} C_VEL
LIN {X 0,Y 601.403,Z 429.527,A -85,B 0,C 180,E1 -792.314,E2 -792.314} C_VEL
LIN {X 0,Y 601.367,Z 440.118,A -85,B 0,C 180,E1 -795.103,E2 -795.103} C_VEL
LIN {X 0,Y 601.355,Z 450.709,A -85,B 0,C 180,E1 -797.858,E2 -797.858} C_VEL
LIN {X 0,Y 601.383,Z 451.536,A -85,B 0,C 180,E1 -798.072,E2 -798.072} C_VEL
LIN {X 0,Y 601.599,Z 465.99,A -85,B 0,C 180,E1 -798.376,E2 -798.376} C_VEL
LIN {X 0,Y 601.512,Z 478.292,A -85,B 0,C 180,E1 -798.763,E2 -798.763} C_VEL
LIN {X 0,Y 601.486,Z 490.953,A -85,B 0,C 180,E1 -799.312,E2 -799.312} C_VEL
LIN {X 0,Y 601.474,Z 501.604,A -85,B 0,C 180,E1 -799.907,E2 -799.907} C_VEL
LIN {X 0,Y 601.449,Z 512.493,A -85,B 0,C 180,E1 -800.671,E2 -800.671} C_VEL
LIN {X 0,Y 601.428,Z 523.127,A -85,B 0,C 180,E1 -801.602,E2 -801.602} C_VEL
LIN {X 0,Y 601.417,Z 530.973,A -85,B 0,C 180,E1 -802.447,E2 -802.447} C_VEL
LIN {X 0,Y 601.369,Z 538.232,A -85,B 0,C 180,E1 -803.399,E2 -803.399} C_VEL
LIN {X 0,Y 601.372,Z 543.874,A -85,B 0,C 180,E1 -804.3,E2 -804.3} C_VEL
LIN {X 0,Y 601.336,Z 548.956,A -85,B 0,C 180,E1 -805.309,E2 -805.309} C_VEL
LIN {X 0,Y 601.368,Z 552.901,A -85,B 0,C 180,E1 -806.316,E2 -806.316} C_VEL
LIN {X 0,Y 601.325,Z 555.812,A -85,B 0,C 180,E1 -807.322,E2 -807.322} C_VEL
LIN {X 0,Y 601.343,Z 557.204,A -85,B 0,C 180,E1 -807.992,E2 -807.992} C_VEL
LIN {X 0,Y 601.339,Z 558.784,A -85,B 0,C 180,E1 -809.332,E2 -809.332} C_VEL
LIN {X 0,Y 601.335,Z 559,A -85,B 0,C 180,E1 -810.001,E2 -810.001} C_VEL
LIN {X 0,Y 601.347,Z 558.183,A -85,B 0,C 180,E1 -811.341,E2 -811.341} C_VEL
LIN {X 0,Y 601.343,Z 557.2,A -85,B 0,C 180,E1 -812.011,E2 -812.011} C_VEL
LIN {X 0,Y 601.325,Z 555.806,A -85,B 0,C 180,E1 -812.681,E2 -812.681} C_VEL
LIN {X 0,Y 601.368,Z 552.892,A -85,B 0,C 180,E1 -813.687,E2 -813.687} C_VEL
LIN {X 0,Y 601.336,Z 548.945,A -85,B 0,C 180,E1 -814.694,E2 -814.694} C_VEL
LIN {X 0,Y 601.372,Z 542.87,A -85,B 0,C 180,E1 -815.87,E2 -815.87} C_VEL
LIN {X 0,Y 601.383,Z 536.227,A -85,B 0,C 180,E1 -816.881,E2 -816.881} C_VEL
LIN {X 0,Y 601.401,Z 527.979,A -85,B 0,C 180,E1 -817.893,E2 -817.893} C_VEL
LIN {X 0,Y 601.436,Z 519.524,A -85,B 0,C 180,E1 -818.739,E2 -818.739} C_VEL
LIN {X 0,Y 601.451,Z 509.076,A -85,B 0,C 180,E1 -819.586,E2 -819.586} C_VEL
LIN {X 0,Y 601.489,Z 498.738,A -85,B 0,C 180,E1 -820.265,E2 -820.265} C_VEL
LIN {X 0,Y 601.486,Z 487.189,A -85,B 0,C 180,E1 -820.871,E2 -820.871} C_VEL
LIN {X 0,Y 601.528,Z 474.299,A -85,B 0,C 180,E1 -821.377,E2 -821.377} C_VEL
LIN {X 0,Y 601.601,Z 461.393,A -85,B 0,C 180,E1 -821.734,E2 -821.734} C_VEL
LIN {X 0,Y 601.383,Z 451.526,A -85,B 0,C 180,E1 -821.93,E2 -821.93} C_VEL
LIN {X 0,Y 601.385,Z 441.432,A -85,B 0,C 180,E1 -824.553,E2 -824.553} C_VEL
LIN {X 0,Y 601.391,Z 430.841,A -85,B 0,C 180,E1 -827.338,E2 -827.338} C_VEL
LIN {X 0,Y 601.429,Z 420.25,A -85,B 0,C 180,E1 -830.166,E2 -830.166} C_VEL
LIN {X 0,Y 601.416,Z 410.983,A -85,B 0,C 180,E1 -832.684,E2 -832.684} C_VEL
LIN {X 0,Y 601.433,Z 401.715,A -85,B 0,C 180,E1 -835.248,E2 -835.248} C_VEL
LIN {X 0,Y 601.5,Z 392.448,A -85,B 0,C 180,E1 -837.864,E2 -837.864} C_VEL
LIN {X 0,Y 601.47,Z 383.181,A -85,B 0,C 180,E1 -840.55,E2 -840.55} C_VEL
LIN {X 0,Y 601.517,Z 375.837,A -85,B 0,C 180,E1 -842.729,E2 -842.729} C_VEL
LIN {X 0,Y 601.589,Z 367.917,A -85,B 0,C 180,E1 -845.138,E2 -845.138} C_VEL
LIN {X 0,Y 601.431,Z 365.572,A -85,B 0,C 180,E1 -845.932,E2 -845.932} C_VEL
LIN {X 0,Y 601.419,Z 365.573,A -85,B 0,C 180,E1 -848.469,E2 -848.469} C_VEL
LIN {X 0,Y 601.415,Z 365.572,A -85,B 0,C 180,E1 -850.875,E2 -850.875} C_VEL
LIN {X 0,Y 601.433,Z 365.571,A -85,B 0,C 180,E1 -853.586,E2 -853.586} C_VEL
LIN {X 0,Y 601.433,Z 365.572,A -85,B 0,C 180,E1 -856.428,E2 -856.428} C_VEL
LIN {X 0,Y 601.418,Z 365.573,A -85,B 0,C 180,E1 -859.427,E2 -859.427} C_VEL
LIN {X 0,Y 601.419,Z 365.574,A -85,B 0,C 180,E1 -861.732,E2 -861.732} C_VEL
LIN {X 0,Y 601.389,Z 365.575,A -85,B 0,C 180,E1 -864.245,E2 -864.245} C_VEL
LIN {X 0,Y 601.419,Z 365.572,A -85,B 0,C 180,E1 -866.686,E2 -866.686} C_VEL
LIN {X 0,Y 601.419,Z 365.574,A -85,B 0,C 180,E1 -869.058,E2 -869.058} C_VEL
LIN {X 0,Y 601.435,Z 365.57,A -85,B 0,C 180,E1 -871.373,E2 -871.373} C_VEL
LIN {X 0,Y 601.414,Z 365.575,A -85,B 0,C 180,E1 -874.133,E2 -874.133} C_VEL
LIN {X 0,Y 601.421,Z 365.572,A -85,B 0,C 180,E1 -876.59,E2 -876.59} C_VEL
LIN {X 0,Y 601.432,Z 365.572,A -85,B 0,C 180,E1 -879.478,E2 -879.478} C_VEL
LIN {X 0,Y 601.396,Z 365.576,A -85,B 0,C 180,E1 -882.312,E2 -882.312} C_VEL
LIN {X 0,Y 601.413,Z 365.574,A -85,B 0,C 180,E1 -884.409,E2 -884.409} C_VEL
LIN {X 0,Y 601.426,Z 365.57,A -85,B 0,C 180,E1 -887.172,E2 -887.172} C_VEL
LIN {X 0,Y 601.429,Z 365.571,A -85,B 0,C 180,E1 -889.905,E2 -889.905} C_VEL
LIN {X 0,Y 601.443,Z 365.57,A -85,B 0,C 180,E1 -892.615,E2 -892.615} C_VEL
LIN {X 0,Y 601.419,Z 365.572,A -85,B 0,C 180,E1 -895.308,E2 -895.308} C_VEL
LIN {X 0,Y 601.434,Z 365.572,A -85,B 0,C 180,E1 -897.991,E2 -897.991} C_VEL
LIN {X 0,Y 601.446,Z 365.568,A -85,B 0,C 180,E1 -900.669,E2 -900.669} C_VEL
LIN {X 0,Y 601.433,Z 365.571,A -85,B 0,C 180,E1 -903.349,E2 -903.349} C_VEL
LIN {X 0,Y 601.407,Z 365.574,A -85,B 0,C 180,E1 -906.037,E2 -906.037} C_VEL
LIN {X 0,Y 601.442,Z 365.569,A -85,B 0,C 180,E1 -908.737,E2 -908.737} C_VEL
LIN {X 0,Y 601.437,Z 365.572,A -85,B 0,C 180,E1 -911.458,E2 -911.458} C_VEL
LIN {X 0,Y 601.41,Z 365.572,A -85,B 0,C 180,E1 -912.376,E2 -912.376} C_VEL
LIN {X 0,Y 600.748,Z 365.655,A -85,B 0,C 180,E1 -912.936,E2 -912.936} C_VEL
LIN {X 0,Y 597.9,Z 366.01,A -85,B 0,C 180,E1 -913.844,E2 -913.844} C_VEL
LIN {X 0,Y 595.488,Z 366.313,A -85,B 0,C 180,E1 -914.574,E2 -914.574} C_VEL
LIN {X 0,Y 594.448,Z 366.44,A -85,B 0,C 180,E1 -915.137,E2 -915.137} C_VEL
LIN {X 0,Y 594.361,Z 366.45,A -85,B 0,C 180,E1 -915.328,E2 -915.328} C_VEL
LIN {X 0,Y 594.352,Z 366.453,A -85,B 0,C 180,E1 -917.905,E2 -917.905} C_VEL
LIN {X 0,Y 594.405,Z 366.448,A -85,B 0,C 180,E1 -920.776,E2 -920.776} C_VEL
LIN {X 0,Y 594.392,Z 366.448,A -85,B 0,C 180,E1 -923.704,E2 -923.704} C_VEL
LIN {X 0,Y 594.388,Z 366.447,A -85,B 0,C 180,E1 -926.699,E2 -926.699} C_VEL
LIN {X 0,Y 594.384,Z 366.449,A -85,B 0,C 180,E1 -928.998,E2 -928.998} C_VEL
LIN {X 0,Y 594.381,Z 366.448,A -85,B 0,C 180,E1 -931.643,E2 -931.643} C_VEL
LIN {X 0,Y 594.382,Z 366.449,A -85,B 0,C 180,E1 -934.58,E2 -934.58} C_VEL
LIN {X 0,Y 594.391,Z 366.448,A -85,B 0,C 180,E1 -937.608,E2 -937.608} C_VEL
LIN {X 0,Y 594.368,Z 366.452,A -85,B 0,C 180,E1 -940.567,E2 -940.567} C_VEL
LIN {X 0,Y 594.369,Z 366.45,A -85,B 0,C 180,E1 -943.299,E2 -943.299} C_VEL
LIN {X 0,Y 594.365,Z 366.45,A -85,B 0,C 180,E1 -946.161,E2 -946.161} C_VEL
LIN {X 0,Y 594.386,Z 366.448,A -85,B 0,C 180,E1 -948.536,E2 -948.536} C_VEL
LIN {X 0,Y 594.384,Z 366.448,A -85,B 0,C 180,E1 -951.296,E2 -951.296} C_VEL
LIN {X 0,Y 594.357,Z 366.452,A -85,B 0,C 180,E1 -953.755,E2 -953.755} C_VEL
LIN {X 0,Y 594.383,Z 366.449,A -85,B 0,C 180,E1 -956.238,E2 -956.238} C_VEL
LIN {X 0,Y 594.382,Z 366.448,A -85,B 0,C 180,E1 -958.65,E2 -958.65} C_VEL
LIN {X 0,Y 594.388,Z 366.449,A -85,B 0,C 180,E1 -961.042,E2 -961.042} C_VEL
LIN {X 0,Y 594.391,Z 366.447,A -85,B 0,C 180,E1 -963.977,E2 -963.977} C_VEL
LIN {X 0,Y 594.391,Z 366.449,A -85,B 0,C 180,E1 -966.295,E2 -966.295} C_VEL
LIN {X 0,Y 594.408,Z 366.445,A -85,B 0,C 180,E1 -969.224,E2 -969.224} C_VEL
LIN {X 0,Y 594.359,Z 366.451,A -85,B 0,C 180,E1 -972.094,E2 -972.094} C_VEL
LIN {X 0,Y 594.372,Z 366.449,A -85,B 0,C 180,E1 -974.218,E2 -974.218} C_VEL
LIN {X 0,Y 594.37,Z 366.45,A -85,B 0,C 180,E1 -977.016,E2 -977.016} C_VEL
LIN {X 0,Y 594.3,Z 366.645,A -85,B 0,C 180,E1 -978.401,E2 -978.401} C_VEL
LIN {X 0,Y 594.287,Z 369.096,A -85,B 0,C 180,E1 -980.469,E2 -980.469} C_VEL
LIN {X 0,Y 594.283,Z 371.544,A -85,B 0,C 180,E1 -982.524,E2 -982.524} C_VEL
LIN {X 0,Y 594.256,Z 373.865,A -85,B 0,C 180,E1 -984.57,E2 -984.57} C_VEL
LIN {X 0,Y 594.233,Z 376.401,A -85,B 0,C 180,E1 -986.609,E2 -986.609} C_VEL
LIN {X 0,Y 594.224,Z 379.008,A -85,B 0,C 180,E1 -988.643,E2 -988.643} C_VEL
LIN {X 0,Y 594.219,Z 381.655,A -85,B 0,C 180,E1 -990.676,E2 -990.676} C_VEL
LIN {X 0,Y 594.207,Z 385.246,A -85,B 0,C 180,E1 -993.389,E2 -993.389} C_VEL
LIN {X 0,Y 594.235,Z 388.907,A -85,B 0,C 180,E1 -996.109,E2 -996.109} C_VEL
LIN {X 0,Y 594.184,Z 392.645,A -85,B 0,C 180,E1 -998.844,E2 -998.844} C_VEL
LIN {X 0,Y 594.205,Z 395.673,A -85,B 0,C 180,E1 -1001.036,E2 -1001.036} C_VEL
LIN {X 0,Y 594.658,Z 400.855,A -85,B 0,C 180,E1 -1001.16,E2 -1001.16} C_VEL
LIN {X 0,Y 594.621,Z 413.359,A -85,B 0,C 180,E1 -1001.503,E2 -1001.503} C_VEL
LIN {X 0,Y 594.526,Z 424.738,A -85,B 0,C 180,E1 -1001.937,E2 -1001.937} C_VEL
LIN {X 0,Y 594.446,Z 436.865,A -85,B 0,C 180,E1 -1002.546,E2 -1002.546} C_VEL
LIN {X 0,Y 594.442,Z 447.667,A -85,B 0,C 180,E1 -1003.241,E2 -1003.241} C_VEL
LIN {X 0,Y 594.398,Z 457.96,A -85,B 0,C 180,E1 -1004.064,E2 -1004.064} C_VEL
LIN {X 0,Y 594.339,Z 466.551,A -85,B 0,C 180,E1 -1004.902,E2 -1004.902} C_VEL
LIN {X 0,Y 594.321,Z 473.998,A -85,B 0,C 180,E1 -1005.78,E2 -1005.78} C_VEL
LIN {X 0,Y 594.309,Z 480.372,A -85,B 0,C 180,E1 -1006.691,E2 -1006.691} C_VEL
LIN {X 0,Y 594.286,Z 485.326,A -85,B 0,C 180,E1 -1007.55,E2 -1007.55} C_VEL
LIN {X 0,Y 594.279,Z 490.299,A -85,B 0,C 180,E1 -1008.619,E2 -1008.619} C_VEL
LIN {X 0,Y 594.238,Z 494.086,A -85,B 0,C 180,E1 -1009.696,E2 -1009.696} C_VEL
LIN {X 0,Y 594.246,Z 496.98,A -85,B 0,C 180,E1 -1010.882,E2 -1010.882} C_VEL
LIN {X 0,Y 594.224,Z 497.973,A -85,B 0,C 180,E1 -1011.507,E2 -1011.507} C_VEL
LIN {X 0,Y 594.239,Z 498.928,A -85,B 0,C 180,E1 -1012.706,E2 -1012.706} C_VEL
LIN {X 0,Y 594.223,Z 498.793,A -85,B 0,C 180,E1 -1013.709,E2 -1013.709} C_VEL
LIN {X 0,Y 594.235,Z 498.126,A -85,B 0,C 180,E1 -1014.451,E2 -1014.451} C_VEL
LIN {X 0,Y 594.221,Z 496.997,A -85,B 0,C 180,E1 -1015.198,E2 -1015.198} C_VEL
LIN {X 0,Y 594.25,Z 494.299,A -85,B 0,C 180,E1 -1016.325,E2 -1016.325} C_VEL
LIN {X 0,Y 594.261,Z 490.165,A -85,B 0,C 180,E1 -1017.503,E2 -1017.503} C_VEL
LIN {X 0,Y 594.256,Z 485.08,A -85,B 0,C 180,E1 -1018.587,E2 -1018.587} C_VEL
LIN {X 0,Y 594.294,Z 477.876,A -85,B 0,C 180,E1 -1019.779,E2 -1019.779} C_VEL
LIN {X 0,Y 594.36,Z 470.39,A -85,B 0,C 180,E1 -1020.755,E2 -1020.755} C_VEL
LIN {X 0,Y 594.394,Z 461.422,A -85,B 0,C 180,E1 -1021.707,E2 -1021.707} C_VEL
LIN {X 0,Y 594.423,Z 451.785,A -85,B 0,C 180,E1 -1022.542,E2 -1022.542} C_VEL
LIN {X 0,Y 594.452,Z 441.8,A -85,B 0,C 180,E1 -1023.246,E2 -1023.246} C_VEL
LIN {X 0,Y 594.541,Z 430.251,A -85,B 0,C 180,E1 -1023.894,E2 -1023.894} C_VEL
LIN {X 0,Y 594.587,Z 417.783,A -85,B 0,C 180,E1 -1024.434,E2 -1024.434} C_VEL
LIN {X 0,Y 594.642,Z 405.09,A -85,B 0,C 180,E1 -1024.83,E2 -1024.83} C_VEL
LIN {X 0,Y 594.477,Z 397.364,A -85,B 0,C 180,E1 -1025.004,E2 -1025.004} C_VEL
LIN {X 0,Y 594.237,Z 395.675,A -85,B 0,C 180,E1 -1025.051,E2 -1025.051} C_VEL
LIN {X 0,Y 594.234,Z 391.678,A -85,B 0,C 180,E1 -1027.95,E2 -1027.95} C_VEL
LIN {X 0,Y 594.21,Z 387.795,A -85,B 0,C 180,E1 -1030.803,E2 -1030.803} C_VEL
LIN {X 0,Y 594.246,Z 384.436,A -85,B 0,C 180,E1 -1033.308,E2 -1033.308} C_VEL
LIN {X 0,Y 594.249,Z 381.211,A -85,B 0,C 180,E1 -1035.751,E2 -1035.751} C_VEL
LIN {X 0,Y 594.238,Z 378.084,A -85,B 0,C 180,E1 -1038.164,E2 -1038.164} C_VEL
LIN {X 0,Y 594.253,Z 375.352,A -85,B 0,C 180,E1 -1040.31,E2 -1040.31} C_VEL
LIN {X 0,Y 594.268,Z 372.411,A -85,B 0,C 180,E1 -1042.905,E2 -1042.905} C_VEL
LIN {X 0,Y 594.321,Z 368.898,A -85,B 0,C 180,E1 -1045.866,E2 -1045.866} C_VEL
LIN {X 0,Y 594.285,Z 366.529,A -85,B 0,C 180,E1 -1047.848,E2 -1047.848} C_VEL
LIN {X 0,Y 594.37,Z 366.448,A -85,B 0,C 180,E1 -1050.223,E2 -1050.223} C_VEL
LIN {X 0,Y 594.372,Z 366.45,A -85,B 0,C 180,E1 -1052.539,E2 -1052.539} C_VEL
LIN {X 0,Y 594.358,Z 366.451,A -85,B 0,C 180,E1 -1054.806,E2 -1054.806} C_VEL
LIN {X 0,Y 594.388,Z 366.446,A -85,B 0,C 180,E1 -1057.254,E2 -1057.254} C_VEL
LIN {X 0,Y 594.363,Z 366.448,A -85,B 0,C 180,E1 -1059.946,E2 -1059.946} C_VEL
LIN {X 0,Y 594.365,Z 366.45,A -85,B 0,C 180,E1 -1062.095,E2 -1062.095} C_VEL
LIN {X 0,Y 594.355,Z 366.451,A -85,B 0,C 180,E1 -1064.219,E2 -1064.219} C_VEL
LIN {X 0,Y 594.366,Z 366.448,A -85,B 0,C 180,E1 -1066.321,E2 -1066.321} C_VEL
LIN {X 0,Y 594.371,Z 366.448,A -85,B 0,C 180,E1 -1069.095,E2 -1069.095} C_VEL
LIN {X 0,Y 594.397,Z 366.444,A -85,B 0,C 180,E1 -1071.843,E2 -1071.843} C_VEL
LIN {X 0,Y 594.39,Z 366.445,A -85,B 0,C 180,E1 -1074.572,E2 -1074.572} C_VEL
LIN {X 0,Y 594.399,Z 366.444,A -85,B 0,C 180,E1 -1077.289,E2 -1077.289} C_VEL
LIN {X 0,Y 594.388,Z 366.445,A -85,B 0,C 180,E1 -1080,E2 -1080} C_VEL
LIN {X 0,Y 594.403,Z 366.443,A -85,B 0,C 180,E1 -1082.711,E2 -1082.711} C_VEL
LIN {X 0,Y 594.379,Z 366.446,A -85,B 0,C 180,E1 -1085.428,E2 -1085.428} C_VEL
LIN {X 0,Y 594.397,Z 366.444,A -85,B 0,C 180,E1 -1088.157,E2 -1088.157} C_VEL
LIN {X 0,Y 594.383,Z 366.446,A -85,B 0,C 180,E1 -1091.083,E2 -1091.083} C_VEL
LIN {X 0,Y 594.364,Z 366.448,A -85,B 0,C 180,E1 -1093.679,E2 -1093.679} C_VEL
LIN {X 0,Y 594.393,Z 366.445,A -85,B 0,C 180,E1 -1096.486,E2 -1096.486} C_VEL
LIN {X 0,Y 594.362,Z 366.45,A -85,B 0,C 180,E1 -1099.335,E2 -1099.335} C_VEL
LIN {X 0,Y 594.353,Z 366.45,A -85,B 0,C 180,E1 -1101.504,E2 -1101.504} C_VEL
LIN {X 0,Y 594.384,Z 366.45,A -85,B 0,C 180,E1 -1103.704,E2 -1103.704} C_VEL
LIN {X 0,Y 594.373,Z 366.449,A -85,B 0,C 180,E1 -1106.7,E2 -1106.7} C_VEL
LIN {X 0,Y 594.371,Z 366.451,A -85,B 0,C 180,E1 -1108.999,E2 -1108.999} C_VEL
LIN {X 0,Y 594.38,Z 366.449,A -85,B 0,C 180,E1 -1111.647,E2 -1111.647} C_VEL
LIN {X 0,Y 594.381,Z 366.451,A -85,B 0,C 180,E1 -1114.58,E2 -1114.58} C_VEL
LIN {X 0,Y 594.377,Z 366.449,A -85,B 0,C 180,E1 -1117.088,E2 -1117.088} C_VEL
LIN {X 0,Y 594.352,Z 366.453,A -85,B 0,C 180,E1 -1119.775,E2 -1119.775} C_VEL
LIN {X 0,Y 594.357,Z 366.451,A -85,B 0,C 180,E1 -1122.377,E2 -1122.377} C_VEL
LIN {X 0,Y 594.35,Z 366.453,A -85,B 0,C 180,E1 -1125.193,E2 -1125.193} C_VEL
LIN {X 0,Y 594.355,Z 366.451,A -85,B 0,C 180,E1 -1127.626,E2 -1127.626} C_VEL
LIN {X 0,Y 594.386,Z 366.447,A -85,B 0,C 180,E1 -1130.323,E2 -1130.323} C_VEL
LIN {X 0,Y 594.377,Z 366.448,A -85,B 0,C 180,E1 -1132.915,E2 -1132.915} C_VEL
LIN {X 0,Y 594.448,Z 366.643,A -85,B 0,C 180,E1 -1133.974,E2 -1133.974} C_VEL
LIN {X 0,Y 594.606,Z 372.543,A -85,B 0,C 180,E1 -1135.83,E2 -1135.83} C_VEL
LIN {X 0,Y 594.573,Z 381.867,A -85,B 0,C 180,E1 -1138.664,E2 -1138.664} C_VEL
LIN {X 0,Y 594.461,Z 391.157,A -85,B 0,C 180,E1 -1141.401,E2 -1141.401} C_VEL
LIN {X 0,Y 594.488,Z 400.402,A -85,B 0,C 180,E1 -1144.063,E2 -1144.063} C_VEL
LIN {X 0,Y 594.427,Z 409.669,A -85,B 0,C 180,E1 -1146.669,E2 -1146.669} C_VEL
LIN {X 0,Y 594.402,Z 418.936,A -85,B 0,C 180,E1 -1149.226,E2 -1149.226} C_VEL
LIN {X 0,Y 594.36,Z 429.527,A -85,B 0,C 180,E1 -1152.097,E2 -1152.097} C_VEL
LIN {X 0,Y 594.304,Z 440.118,A -85,B 0,C 180,E1 -1154.922,E2 -1154.922} C_VEL
LIN {X 0,Y 594.283,Z 450.709,A -85,B 0,C 180,E1 -1157.711,E2 -1157.711} C_VEL
LIN {X 0,Y 594.284,Z 451.654,A -85,B 0,C 180,E1 -1157.941,E2 -1157.941} C_VEL
LIN {X 0,Y 594.689,Z 456.171,A -85,B 0,C 180,E1 -1158.023,E2 -1158.023} C_VEL
LIN {X 0,Y 594.623,Z 469.791,A -85,B 0,C 180,E1 -1158.346,E2 -1158.346} C_VEL
LIN {X 0,Y 594.551,Z 480.762,A -85,B 0,C 180,E1 -1158.725,E2 -1158.725} C_VEL
LIN {X 0,Y 594.491,Z 492.663,A -85,B 0,C 180,E1 -1159.271,E2 -1159.271} C_VEL
LIN {X 0,Y 594.475,Z 504.221,A -85,B 0,C 180,E1 -1159.959,E2 -1159.959} C_VEL
LIN {X 0,Y 594.414,Z 514.613,A -85,B 0,C 180,E1 -1160.731,E2 -1160.731} C_VEL
LIN {X 0,Y 594.382,Z 523.127,A -85,B 0,C 180,E1 -1161.502,E2 -1161.502} C_VEL
LIN {X 0,Y 594.346,Z 530.973,A -85,B 0,C 180,E1 -1162.357,E2 -1162.357} C_VEL
LIN {X 0,Y 594.281,Z 538.819,A -85,B 0,C 180,E1 -1163.409,E2 -1163.409} C_VEL
LIN {X 0,Y 594.289,Z 545.688,A -85,B 0,C 180,E1 -1164.573,E2 -1164.573} C_VEL
LIN {X 0,Y 594.27,Z 550.377,A -85,B 0,C 180,E1 -1165.593,E2 -1165.593} C_VEL
LIN {X 0,Y 594.267,Z 553.96,A -85,B 0,C 180,E1 -1166.611,E2 -1166.611} C_VEL
LIN {X 0,Y 594.226,Z 555.812,A -85,B 0,C 180,E1 -1167.29,E2 -1167.29} C_VEL
LIN {X 0,Y 594.242,Z 557.204,A -85,B 0,C 180,E1 -1167.968,E2 -1167.968} C_VEL
LIN {X 0,Y 594.239,Z 558.785,A -85,B 0,C 180,E1 -1169.324,E2 -1169.324} C_VEL
LIN {X 0,Y 594.236,Z 559,A -85,B 0,C 180,E1 -1170.001,E2 -1170.001} C_VEL
LIN {X 0,Y 594.247,Z 558.183,A -85,B 0,C 180,E1 -1171.357,E2 -1171.357} C_VEL
LIN {X 0,Y 594.242,Z 557.2,A -85,B 0,C 180,E1 -1172.035,E2 -1172.035} C_VEL
LIN {X 0,Y 594.226,Z 555.806,A -85,B 0,C 180,E1 -1172.713,E2 -1172.713} C_VEL
LIN {X 0,Y 594.289,Z 552.892,A -85,B 0,C 180,E1 -1173.731,E2 -1173.731} C_VEL
LIN {X 0,Y 594.241,Z 548.945,A -85,B 0,C 180,E1 -1174.75,E2 -1174.75} C_VEL
LIN {X 0,Y 594.304,Z 542.87,A -85,B 0,C 180,E1 -1175.94,E2 -1175.94} C_VEL
LIN {X 0,Y 594.309,Z 536.227,A -85,B 0,C 180,E1 -1176.963,E2 -1176.963} C_VEL
LIN {X 0,Y 594.36,Z 527.979,A -85,B 0,C 180,E1 -1177.988,E2 -1177.988} C_VEL
LIN {X 0,Y 594.382,Z 519.524,A -85,B 0,C 180,E1 -1178.843,E2 -1178.843} C_VEL
LIN {X 0,Y 594.435,Z 509.077,A -85,B 0,C 180,E1 -1179.7,E2 -1179.7} C_VEL
LIN {X 0,Y 594.464,Z 498.739,A -85,B 0,C 180,E1 -1180.388,E2 -1180.388} C_VEL
LIN {X 0,Y 594.504,Z 486.741,A -85,B 0,C 180,E1 -1181.02,E2 -1181.02} C_VEL
LIN {X 0,Y 594.565,Z 474.456,A -85,B 0,C 180,E1 -1181.506,E2 -1181.506} C_VEL
LIN {X 0,Y 594.654,Z 461.392,A -85,B 0,C 180,E1 -1181.873,E2 -1181.873} C_VEL
LIN {X 0,Y 594.461,Z 452.881,A -85,B 0,C 180,E1 -1182.037,E2 -1182.037} C_VEL
LIN {X 0,Y 594.295,Z 451.526,A -85,B 0,C 180,E1 -1182.075,E2 -1182.075} C_VEL
LIN {X 0,Y 594.313,Z 441.432,A -85,B 0,C 180,E1 -1184.73,E2 -1184.73} C_VEL
LIN {X 0,Y 594.336,Z 430.841,A -85,B 0,C 180,E1 -1187.551,E2 -1187.551} C_VEL
LIN {X 0,Y 594.386,Z 420.25,A -85,B 0,C 180,E1 -1190.415,E2 -1190.415} C_VEL
LIN {X 0,Y 594.404,Z 410.983,A -85,B 0,C 180,E1 -1192.967,E2 -1192.967} C_VEL
LIN {X 0,Y 594.476,Z 401.715,A -85,B 0,C 180,E1 -1195.564,E2 -1195.564} C_VEL
LIN {X 0,Y 594.495,Z 392.448,A -85,B 0,C 180,E1 -1198.222,E2 -1198.222} C_VEL
LIN {X 0,Y 594.529,Z 383.181,A -85,B 0,C 180,E1 -1200.946,E2 -1200.946} C_VEL
LIN {X 0,Y 594.639,Z 375.238,A -85,B 0,C 180,E1 -1203.339,E2 -1203.339} C_VEL
LIN {X 0,Y 594.554,Z 367.295,A -85,B 0,C 180,E1 -1205.812,E2 -1205.812} C_VEL
LIN {X 0,Y 594.377,Z 366.452,A -85,B 0,C 180,E1 -1206.139,E2 -1206.139} C_VEL
LIN {X 0,Y 594.375,Z 366.449,A -85,B 0,C 180,E1 -1208.806,E2 -1208.806} C_VEL
LIN {X 0,Y 594.386,Z 366.448,A -85,B 0,C 180,E1 -1211.848,E2 -1211.848} C_VEL
LIN {X 0,Y 594.364,Z 366.451,A -85,B 0,C 180,E1 -1214.239,E2 -1214.239} C_VEL
LIN {X 0,Y 594.365,Z 366.45,A -85,B 0,C 180,E1 -1217.148,E2 -1217.148} C_VEL
LIN {X 0,Y 594.373,Z 366.45,A -85,B 0,C 180,E1 -1219.433,E2 -1219.433} C_VEL
LIN {X 0,Y 594.394,Z 366.447,A -85,B 0,C 180,E1 -1222.392,E2 -1222.392} C_VEL
LIN {X 0,Y 594.383,Z 366.448,A -85,B 0,C 180,E1 -1225.42,E2 -1225.42} C_VEL
LIN {X 0,Y 594.38,Z 366.448,A -85,B 0,C 180,E1 -1228.358,E2 -1228.358} C_VEL
LIN {X 0,Y 594.387,Z 366.45,A -85,B 0,C 180,E1 -1231.042,E2 -1231.042} C_VEL
LIN {X 0,Y 594.388,Z 366.448,A -85,B 0,C 180,E1 -1233.978,E2 -1233.978} C_VEL
LIN {X 0,Y 594.389,Z 366.45,A -85,B 0,C 180,E1 -1236.296,E2 -1236.296} C_VEL
LIN {X 0,Y 594.408,Z 366.447,A -85,B 0,C 180,E1 -1239.224,E2 -1239.224} C_VEL
LIN {X 0,Y 594.354,Z 366.452,A -85,B 0,C 180,E1 -1242.095,E2 -1242.095} C_VEL
LIN {X 0,Y 594.366,Z 366.45,A -85,B 0,C 180,E1 -1244.219,E2 -1244.219} C_VEL
LIN {X 0,Y 594.382,Z 366.449,A -85,B 0,C 180,E1 -1246.321,E2 -1246.321} C_VEL
LIN {X 0,Y 594.383,Z 366.448,A -85,B 0,C 180,E1 -1249.095,E2 -1249.095} C_VEL
LIN {X 0,Y 594.416,Z 366.446,A -85,B 0,C 180,E1 -1251.843,E2 -1251.843} C_VEL
LIN {X 0,Y 594.393,Z 366.447,A -85,B 0,C 180,E1 -1254.572,E2 -1254.572} C_VEL
LIN {X 0,Y 594.403,Z 366.446,A -85,B 0,C 180,E1 -1257.289,E2 -1257.289} C_VEL
LIN {X 0,Y 594.415,Z 366.446,A -85,B 0,C 180,E1 -1260,E2 -1260} C_VEL
LIN {X 0,Y 594.409,Z 366.445,A -85,B 0,C 180,E1 -1262.711,E2 -1262.711} C_VEL
LIN {X 0,Y 594.398,Z 366.447,A -85,B 0,C 180,E1 -1265.428,E2 -1265.428} C_VEL
LIN {X 0,Y 594.415,Z 366.445,A -85,B 0,C 180,E1 -1268.157,E2 -1268.157} C_VEL
LIN {X 0,Y 594.397,Z 366.446,A -85,B 0,C 180,E1 -1271.076,E2 -1271.076} C_VEL
LIN {X 0,Y 594.381,Z 366.45,A -85,B 0,C 180,E1 -1273.679,E2 -1273.679} C_VEL
LIN {X 0,Y 594.361,Z 366.45,A -85,B 0,C 180,E1 -1275.328,E2 -1275.328} C_VEL
LIN {X 0,Y 593.685,Z 366.536,A -85,B 0,C 180,E1 -1275.894,E2 -1275.894} C_VEL
LIN {X 0,Y 590.818,Z 366.893,A -85,B 0,C 180,E1 -1276.812,E2 -1276.812} C_VEL
LIN {X 0,Y 588.409,Z 367.194,A -85,B 0,C 180,E1 -1277.551,E2 -1277.551} C_VEL
LIN {X 0,Y 587.387,Z 367.319,A -85,B 0,C 180,E1 -1278.121,E2 -1278.121} C_VEL
LIN {X 0,Y 587.31,Z 367.328,A -85,B 0,C 180,E1 -1278.314,E2 -1278.314} C_VEL
LIN {X 0,Y 587.334,Z 367.327,A -85,B 0,C 180,E1 -1281.037,E2 -1281.037} C_VEL
LIN {X 0,Y 587.325,Z 367.327,A -85,B 0,C 180,E1 -1283.259,E2 -1283.259} C_VEL
LIN {X 0,Y 587.333,Z 367.326,A -85,B 0,C 180,E1 -1285.517,E2 -1285.517} C_VEL
LIN {X 0,Y 587.351,Z 367.325,A -85,B 0,C 180,E1 -1287.818,E2 -1287.818} C_VEL
LIN {X 0,Y 587.341,Z 367.325,A -85,B 0,C 180,E1 -1290.51,E2 -1290.51} C_VEL
LIN {X 0,Y 587.332,Z 367.328,A -85,B 0,C 180,E1 -1293.397,E2 -1293.397} C_VEL
LIN {X 0,Y 587.294,Z 367.331,A -85,B 0,C 180,E1 -1295.9,E2 -1295.9} C_VEL
LIN {X 0,Y 587.324,Z 367.33,A -85,B 0,C 180,E1 -1298.48,E2 -1298.48} C_VEL
LIN {X 0,Y 587.338,Z 367.326,A -85,B 0,C 180,E1 -1301.157,E2 -1301.157} C_VEL
LIN {X 0,Y 587.316,Z 367.328,A -85,B 0,C 180,E1 -1304.112,E2 -1304.112} C_VEL
LIN {X 0,Y 587.318,Z 367.329,A -85,B 0,C 180,E1 -1306.993,E2 -1306.993} C_VEL
LIN {X 0,Y 587.321,Z 367.33,A -85,B 0,C 180,E1 -1309.746,E2 -1309.746} C_VEL
LIN {X 0,Y 587.35,Z 367.324,A -85,B 0,C 180,E1 -1312.392,E2 -1312.392} C_VEL
LIN {X 0,Y 587.365,Z 367.323,A -85,B 0,C 180,E1 -1315.779,E2 -1315.779} C_VEL
LIN {X 0,Y 587.348,Z 367.326,A -85,B 0,C 180,E1 -1318.231,E2 -1318.231} C_VEL
LIN {X 0,Y 587.354,Z 367.324,A -85,B 0,C 180,E1 -1320.866,E2 -1320.866} C_VEL
LIN {X 0,Y 587.364,Z 367.322,A -85,B 0,C 180,E1 -1323.818,E2 -1323.818} C_VEL
LIN {X 0,Y 587.339,Z 367.325,A -85,B 0,C 180,E1 -1325.993,E2 -1325.993} C_VEL
LIN {X 0,Y 587.327,Z 367.327,A -85,B 0,C 180,E1 -1328.225,E2 -1328.225} C_VEL
LIN {X 0,Y 587.352,Z 367.324,A -85,B 0,C 180,E1 -1331.15,E2 -1331.15} C_VEL
LIN {X 0,Y 587.327,Z 367.327,A -85,B 0,C 180,E1 -1334.024,E2 -1334.024} C_VEL
LIN {X 0,Y 587.367,Z 367.322,A -85,B 0,C 180,E1 -1336.153,E2 -1336.153} C_VEL
LIN {X 0,Y 587.263,Z 367.337,A -85,B 0,C 180,E1 -1338.26,E2 -1338.26} C_VEL
LIN {X 0,Y 587.224,Z 369.56,A -85,B 0,C 180,E1 -1340.353,E2 -1340.353} C_VEL
LIN {X 0,Y 587.223,Z 372.036,A -85,B 0,C 180,E1 -1342.434,E2 -1342.434} C_VEL
LIN {X 0,Y 587.182,Z 374.38,A -85,B 0,C 180,E1 -1344.504,E2 -1344.504} C_VEL
LIN {X 0,Y 587.16,Z 376.781,A -85,B 0,C 180,E1 -1346.568,E2 -1346.568} C_VEL
LIN {X 0,Y 587.136,Z 379.388,A -85,B 0,C 180,E1 -1348.627,E2 -1348.627} C_VEL
LIN {X 0,Y 587.128,Z 382.034,A -85,B 0,C 180,E1 -1350.685,E2 -1350.685} C_VEL
LIN {X 0,Y 587.134,Z 385.626,A -85,B 0,C 180,E1 -1353.43,E2 -1353.43} C_VEL
LIN {X 0,Y 587.139,Z 389.761,A -85,B 0,C 180,E1 -1356.534,E2 -1356.534} C_VEL
LIN {X 0,Y 587.09,Z 393.029,A -85,B 0,C 180,E1 -1358.951,E2 -1358.951} C_VEL
LIN {X 0,Y 587.115,Z 395.814,A -85,B 0,C 180,E1 -1360.904,E2 -1360.904} C_VEL
LIN {X 0,Y 587.715,Z 401.338,A -85,B 0,C 180,E1 -1361.029,E2 -1361.029} C_VEL
LIN {X 0,Y 587.666,Z 414.175,A -85,B 0,C 180,E1 -1361.392,E2 -1361.392} C_VEL
LIN {X 0,Y 587.523,Z 427.059,A -85,B 0,C 180,E1 -1361.907,E2 -1361.907} C_VEL
LIN {X 0,Y 587.44,Z 438.585,A -85,B 0,C 180,E1 -1362.522,E2 -1362.522} C_VEL
LIN {X 0,Y 587.412,Z 450.234,A -85,B 0,C 180,E1 -1363.314,E2 -1363.314} C_VEL
LIN {X 0,Y 587.332,Z 459.938,A -85,B 0,C 180,E1 -1364.133,E2 -1364.133} C_VEL
LIN {X 0,Y 587.29,Z 469.048,A -85,B 0,C 180,E1 -1365.085,E2 -1365.085} C_VEL
LIN {X 0,Y 587.254,Z 477.343,A -85,B 0,C 180,E1 -1366.154,E2 -1366.154} C_VEL
LIN {X 0,Y 587.225,Z 483.889,A -85,B 0,C 180,E1 -1367.211,E2 -1367.211} C_VEL
LIN {X 0,Y 587.171,Z 488.467,A -85,B 0,C 180,E1 -1368.13,E2 -1368.13} C_VEL
LIN {X 0,Y 587.176,Z 491.912,A -85,B 0,C 180,E1 -1368.992,E2 -1368.992} C_VEL
LIN {X 0,Y 587.156,Z 495.83,A -85,B 0,C 180,E1 -1370.309,E2 -1370.309} C_VEL
LIN {X 0,Y 587.141,Z 497.292,A -85,B 0,C 180,E1 -1371.043,E2 -1371.043} C_VEL
LIN {X 0,Y 587.139,Z 498.306,A -85,B 0,C 180,E1 -1371.78,E2 -1371.78} C_VEL
LIN {X 0,Y 587.125,Z 498.956,A -85,B 0,C 180,E1 -1372.823,E2 -1372.823} C_VEL
LIN {X 0,Y 587.123,Z 498.591,A -85,B 0,C 180,E1 -1374.014,E2 -1374.014} C_VEL
LIN {X 0,Y 587.145,Z 497.742,A -85,B 0,C 180,E1 -1374.766,E2 -1374.766} C_VEL
LIN {X 0,Y 587.139,Z 494.915,A -85,B 0,C 180,E1 -1376.137,E2 -1376.137} C_VEL
LIN {X 0,Y 587.173,Z 490.986,A -85,B 0,C 180,E1 -1377.354,E2 -1377.354} C_VEL
LIN {X 0,Y 587.171,Z 485.348,A -85,B 0,C 180,E1 -1378.603,E2 -1378.603} C_VEL
LIN {X 0,Y 587.212,Z 478.407,A -85,B 0,C 180,E1 -1379.779,E2 -1379.779} C_VEL
LIN {X 0,Y 587.289,Z 470.516,A -85,B 0,C 180,E1 -1380.834,E2 -1380.834} C_VEL
LIN {X 0,Y 587.337,Z 461.197,A -85,B 0,C 180,E1 -1381.834,E2 -1381.834} C_VEL
LIN {X 0,Y 587.406,Z 451.701,A -85,B 0,C 180,E1 -1382.664,E2 -1382.664} C_VEL
LIN {X 0,Y 587.429,Z 441.502,A -85,B 0,C 180,E1 -1383.388,E2 -1383.388} C_VEL
LIN {X 0,Y 587.541,Z 429.745,A -85,B 0,C 180,E1 -1384.05,E2 -1384.05} C_VEL
LIN {X 0,Y 587.637,Z 417.342,A -85,B 0,C 180,E1 -1384.587,E2 -1384.587} C_VEL
LIN {X 0,Y 587.681,Z 404.804,A -85,B 0,C 180,E1 -1384.979,E2 -1384.979} C_VEL
LIN {X 0,Y 587.488,Z 397.976,A -85,B 0,C 180,E1 -1385.137,E2 -1385.137} C_VEL
LIN {X 0,Y 587.127,Z 395.66,A -85,B 0,C 180,E1 -1385.21,E2 -1385.21} C_VEL
LIN {X 0,Y 587.128,Z 392.115,A -85,B 0,C 180,E1 -1387.812,E2 -1387.812} C_VEL
LIN {X 0,Y 587.133,Z 388.808,A -85,B 0,C 180,E1 -1390.267,E2 -1390.267} C_VEL
LIN {X 0,Y 587.175,Z 385.039,A -85,B 0,C 180,E1 -1393.103,E2 -1393.103} C_VEL
LIN {X 0,Y 587.168,Z 381.219,A -85,B 0,C 180,E1 -1396.035,E2 -1396.035} C_VEL
LIN {X 0,Y 587.137,Z 377.658,A -85,B 0,C 180,E1 -1398.826,E2 -1398.826} C_VEL
LIN {X 0,Y 587.166,Z 374.612,A -85,B 0,C 180,E1 -1401.508,E2 -1401.508} C_VEL
LIN {X 0,Y 587.22,Z 371.187,A -85,B 0,C 180,E1 -1404.469,E2 -1404.469} C_VEL
LIN {X 0,Y 587.229,Z 368.277,A -85,B 0,C 180,E1 -1406.901,E2 -1406.901} C_VEL
LIN {X 0,Y 587.273,Z 367.337,A -85,B 0,C 180,E1 -1408.171,E2 -1408.171} C_VEL
LIN {X 0,Y 587.337,Z 367.327,A -85,B 0,C 180,E1 -1410.864,E2 -1410.864} C_VEL
LIN {X 0,Y 587.342,Z 367.327,A -85,B 0,C 180,E1 -1413.817,E2 -1413.817} C_VEL
LIN {X 0,Y 587.36,Z 367.322,A -85,B 0,C 180,E1 -1416.743,E2 -1416.743} C_VEL
LIN {X 0,Y 587.318,Z 367.326,A -85,B 0,C 180,E1 -1419.695,E2 -1419.695} C_VEL
LIN {X 0,Y 587.318,Z 367.33,A -85,B 0,C 180,E1 -1421.873,E2 -1421.873} C_VEL
LIN {X 0,Y 587.31,Z 367.327,A -85,B 0,C 180,E1 -1424.024,E2 -1424.024} C_VEL
LIN {X 0,Y 587.349,Z 367.324,A -85,B 0,C 180,E1 -1426.154,E2 -1426.154} C_VEL
LIN {X 0,Y 587.333,Z 367.325,A -85,B 0,C 180,E1 -1428.962,E2 -1428.962} C_VEL
LIN {X 0,Y 587.351,Z 367.322,A -85,B 0,C 180,E1 -1431.745,E2 -1431.745} C_VEL
LIN {X 0,Y 587.356,Z 367.322,A -85,B 0,C 180,E1 -1434.507,E2 -1434.507} C_VEL
LIN {X 0,Y 587.364,Z 367.32,A -85,B 0,C 180,E1 -1437.257,E2 -1437.257} C_VEL
LIN {X 0,Y 587.357,Z 367.321,A -85,B 0,C 180,E1 -1440,E2 -1440} C_VEL
LIN {X 0,Y 587.368,Z 367.32,A -85,B 0,C 180,E1 -1442.743,E2 -1442.743} C_VEL
LIN {X 0,Y 587.344,Z 367.323,A -85,B 0,C 180,E1 -1445.493,E2 -1445.493} C_VEL
LIN {X 0,Y 587.35,Z 367.322,A -85,B 0,C 180,E1 -1448.256,E2 -1448.256} C_VEL
LIN {X 0,Y 587.36,Z 367.321,A -85,B 0,C 180,E1 -1451.151,E2 -1451.151} C_VEL
LIN {X 0,Y 587.344,Z 367.327,A -85,B 0,C 180,E1 -1454.262,E2 -1454.262} C_VEL
LIN {X 0,Y 587.34,Z 367.324,A -85,B 0,C 180,E1 -1457.406,E2 -1457.406} C_VEL
LIN {X 0,Y 587.334,Z 367.327,A -85,B 0,C 180,E1 -1459.575,E2 -1459.575} C_VEL
LIN {X 0,Y 587.353,Z 367.325,A -85,B 0,C 180,E1 -1462.513,E2 -1462.513} C_VEL
LIN {X 0,Y 587.319,Z 367.327,A -85,B 0,C 180,E1 -1465.518,E2 -1465.518} C_VEL
LIN {X 0,Y 587.333,Z 367.329,A -85,B 0,C 180,E1 -1467.819,E2 -1467.819} C_VEL
LIN {X 0,Y 587.325,Z 367.33,A -85,B 0,C 180,E1 -1470.512,E2 -1470.512} C_VEL
LIN {X 0,Y 587.324,Z 367.329,A -85,B 0,C 180,E1 -1473.114,E2 -1473.114} C_VEL
LIN {X 0,Y 587.344,Z 367.327,A -85,B 0,C 180,E1 -1475.897,E2 -1475.897} C_VEL
LIN {X 0,Y 587.313,Z 367.33,A -85,B 0,C 180,E1 -1478.481,E2 -1478.481} C_VEL
LIN {X 0,Y 587.35,Z 367.325,A -85,B 0,C 180,E1 -1481.156,E2 -1481.156} C_VEL
LIN {X 0,Y 587.313,Z 367.331,A -85,B 0,C 180,E1 -1484.115,E2 -1484.115} C_VEL
LIN {X 0,Y 587.308,Z 367.33,A -85,B 0,C 180,E1 -1486.996,E2 -1486.996} C_VEL
LIN {X 0,Y 587.319,Z 367.328,A -85,B 0,C 180,E1 -1489.749,E2 -1489.749} C_VEL
LIN {X 0,Y 587.336,Z 367.327,A -85,B 0,C 180,E1 -1492.394,E2 -1492.394} C_VEL
LIN {X 0,Y 587.376,Z 367.47,A -85,B 0,C 180,E1 -1493.737,E2 -1493.737} C_VEL
LIN {X 0,Y 587.671,Z 371.277,A -85,B 0,C 180,E1 -1494.97,E2 -1494.97} C_VEL
LIN {X 0,Y 587.589,Z 379.22,A -85,B 0,C 180,E1 -1497.439,E2 -1497.439} C_VEL
LIN {X 0,Y 587.534,Z 387.163,A -85,B 0,C 180,E1 -1499.843,E2 -1499.843} C_VEL
LIN {X 0,Y 587.461,Z 396.573,A -85,B 0,C 180,E1 -1502.619,E2 -1502.619} C_VEL
LIN {X 0,Y 587.44,Z 405.697,A -85,B 0,C 180,E1 -1505.247,E2 -1505.247} C_VEL
LIN {X 0,Y 587.387,Z 416.288,A -85,B 0,C 180,E1 -1508.23,E2 -1508.23} C_VEL
LIN {X 0,Y 587.31,Z 426.879,A -85,B 0,C 180,E1 -1511.152,E2 -1511.152} C_VEL
LIN {X 0,Y 587.261,Z 437.47,A -85,B 0,C 180,E1 -1514.025,E2 -1514.025} C_VEL
LIN {X 0,Y 587.232,Z 448.061,A -85,B 0,C 180,E1 -1516.858,E2 -1516.858} C_VEL
LIN {X 0,Y 587.221,Z 451.578,A -85,B 0,C 180,E1 -1517.791,E2 -1517.791} C_VEL
LIN {X 0,Y 587.73,Z 457.313,A -85,B 0,C 180,E1 -1517.901,E2 -1517.901} C_VEL
LIN {X 0,Y 587.68,Z 470.551,A -85,B 0,C 180,E1 -1518.228,E2 -1518.228} C_VEL
LIN {X 0,Y 587.567,Z 482.374,A -85,B 0,C 180,E1 -1518.655,E2 -1518.655} C_VEL
LIN {X 0,Y 587.481,Z 494.236,A -85,B 0,C 180,E1 -1519.228,E2 -1519.228} C_VEL
LIN {X 0,Y 587.467,Z 505.499,A -85,B 0,C 180,E1 -1519.925,E2 -1519.925} C_VEL
LIN {X 0,Y 587.384,Z 515.664,A -85,B 0,C 180,E1 -1520.706,E2 -1520.706} C_VEL
LIN {X 0,Y 587.339,Z 524.801,A -85,B 0,C 180,E1 -1521.573,E2 -1521.573} C_VEL
LIN {X 0,Y 587.258,Z 533.703,A -85,B 0,C 180,E1 -1522.61,E2 -1522.61} C_VEL
LIN {X 0,Y 587.195,Z 540.748,A -85,B 0,C 180,E1 -1523.627,E2 -1523.627} C_VEL
LIN {X 0,Y 587.211,Z 545.688,A -85,B 0,C 180,E1 -1524.507,E2 -1524.507} C_VEL
LIN {X 0,Y 587.188,Z 550.377,A -85,B 0,C 180,E1 -1525.539,E2 -1525.539} C_VEL
LIN {X 0,Y 587.193,Z 553.96,A -85,B 0,C 180,E1 -1526.571,E2 -1526.571} C_VEL
LIN {X 0,Y 587.132,Z 555.812,A -85,B 0,C 180,E1 -1527.257,E2 -1527.257} C_VEL
LIN {X 0,Y 587.141,Z 557.204,A -85,B 0,C 180,E1 -1527.943,E2 -1527.943} C_VEL
LIN {X 0,Y 587.14,Z 558.785,A -85,B 0,C 180,E1 -1529.315,E2 -1529.315} C_VEL
LIN {X 0,Y 587.137,Z 559,A -85,B 0,C 180,E1 -1530.001,E2 -1530.001} C_VEL
LIN {X 0,Y 587.147,Z 558.183,A -85,B 0,C 180,E1 -1531.373,E2 -1531.373} C_VEL
LIN {X 0,Y 587.141,Z 557.2,A -85,B 0,C 180,E1 -1532.059,E2 -1532.059} C_VEL
LIN {X 0,Y 587.132,Z 555.806,A -85,B 0,C 180,E1 -1532.746,E2 -1532.746} C_VEL
LIN {X 0,Y 587.213,Z 552.892,A -85,B 0,C 180,E1 -1533.776,E2 -1533.776} C_VEL
LIN {X 0,Y 587.147,Z 548.945,A -85,B 0,C 180,E1 -1534.808,E2 -1534.808} C_VEL
LIN {X 0,Y 587.217,Z 542.87,A -85,B 0,C 180,E1 -1536.012,E2 -1536.012} C_VEL
LIN {X 0,Y 587.246,Z 536.227,A -85,B 0,C 180,E1 -1537.047,E2 -1537.047} C_VEL
LIN {X 0,Y 587.3,Z 527.979,A -85,B 0,C 180,E1 -1538.084,E2 -1538.084} C_VEL
LIN {X 0,Y 587.344,Z 519.524,A -85,B 0,C 180,E1 -1538.95,E2 -1538.95} C_VEL
LIN {X 0,Y 587.421,Z 509.077,A -85,B 0,C 180,E1 -1539.817,E2 -1539.817} C_VEL
LIN {X 0,Y 587.479,Z 498.739,A -85,B 0,C 180,E1 -1540.513,E2 -1540.513} C_VEL
LIN {X 0,Y 587.532,Z 487.133,A -85,B 0,C 180,E1 -1541.135,E2 -1541.135} C_VEL
LIN {X 0,Y 587.626,Z 474.657,A -85,B 0,C 180,E1 -1541.637,E2 -1541.637} C_VEL
LIN {X 0,Y 587.718,Z 461.392,A -85,B 0,C 180,E1 -1542.015,E2 -1542.015} C_VEL
LIN {X 0,Y 587.498,Z 453.538,A -85,B 0,C 180,E1 -1542.173,E2 -1542.173} C_VEL
LIN {X 0,Y 587.205,Z 451.526,A -85,B 0,C 180,E1 -1542.223,E2 -1542.223} C_VEL
LIN {X 0,Y 587.259,Z 441.432,A -85,B 0,C 180,E1 -1544.911,E2 -1544.911} C_VEL
LIN {X 0,Y 587.303,Z 430.841,A -85,B 0,C 180,E1 -1547.768,E2 -1547.768} C_VEL
LIN {X 0,Y 587.378,Z 420.25,A -85,B 0,C 180,E1 -1550.67,E2 -1550.67} C_VEL
LIN {X 0,Y 587.39,Z 410.983,A -85,B 0,C 180,E1 -1553.257,E2 -1553.257} C_VEL
LIN {X 0,Y 587.487,Z 401.83,A -85,B 0,C 180,E1 -1555.858,E2 -1555.858} C_VEL
LIN {X 0,Y 587.468,Z 392.448,A -85,B 0,C 180,E1 -1558.59,E2 -1558.59} C_VEL
LIN {X 0,Y 587.567,Z 384.505,A -85,B 0,C 180,E1 -1560.954,E2 -1560.954} C_VEL
LIN {X 0,Y 587.691,Z 376.562,A -85,B 0,C 180,E1 -1563.375,E2 -1563.375} C_VEL
LIN {X 0,Y 587.591,Z 368.619,A -85,B 0,C 180,E1 -1565.88,E2 -1565.88} C_VEL
LIN {X 0,Y 587.318,Z 367.331,A -85,B 0,C 180,E1 -1566.323,E2 -1566.323} C_VEL
LIN {X 0,Y 587.322,Z 367.328,A -85,B 0,C 180,E1 -1568.94,E2 -1568.94} C_VEL
LIN {X 0,Y 587.34,Z 367.326,A -85,B 0,C 180,E1 -1571.157,E2 -1571.157} C_VEL
LIN {X 0,Y 587.317,Z 367.328,A -85,B 0,C 180,E1 -1574.112,E2 -1574.112} C_VEL
LIN {X 0,Y 587.318,Z 367.328,A -85,B 0,C 180,E1 -1576.994,E2 -1576.994} C_VEL
LIN {X 0,Y 587.316,Z 367.33,A -85,B 0,C 180,E1 -1579.746,E2 -1579.746} C_VEL
LIN {X 0,Y 587.349,Z 367.324,A -85,B 0,C 180,E1 -1582.392,E2 -1582.392} C_VEL
LIN {X 0,Y 587.348,Z 367.325,A -85,B 0,C 180,E1 -1585.653,E2 -1585.653} C_VEL
LIN {X 0,Y 587.345,Z 367.325,A -85,B 0,C 180,E1 -1588.231,E2 -1588.231} C_VEL
LIN {X 0,Y 587.354,Z 367.325,A -85,B 0,C 180,E1 -1590.867,E2 -1590.867} C_VEL
LIN {X 0,Y 587.363,Z 367.322,A -85,B 0,C 180,E1 -1593.819,E2 -1593.819} C_VEL
LIN {X 0,Y 587.329,Z 367.327,A -85,B 0,C 180,E1 -1595.993,E2 -1595.993} C_VEL
LIN {X 0,Y 587.321,Z 367.329,A -85,B 0,C 180,E1 -1598.226,E2 -1598.226} C_VEL
LIN {X 0,Y 587.355,Z 367.324,A -85,B 0,C 180,E1 -1601.151,E2 -1601.151} C_VEL
LIN {X 0,Y 587.325,Z 367.327,A -85,B 0,C 180,E1 -1604.025,E2 -1604.025} C_VEL
LIN {X 0,Y 587.361,Z 367.323,A -85,B 0,C 180,E1 -1606.154,E2 -1606.154} C_VEL
LIN {X 0,Y 587.348,Z 367.324,A -85,B 0,C 180,E1 -1608.962,E2 -1608.962} C_VEL
LIN {X 0,Y 587.371,Z 367.323,A -85,B 0,C 180,E1 -1611.745,E2 -1611.745} C_VEL
LIN {X 0,Y 587.358,Z 367.323,A -85,B 0,C 180,E1 -1614.507,E2 -1614.507} C_VEL
LIN {X 0,Y 587.37,Z 367.322,A -85,B 0,C 180,E1 -1617.257,E2 -1617.257} C_VEL
LIN {X 0,Y 587.384,Z 367.322,A -85,B 0,C 180,E1 -1620,E2 -1620} C_VEL
LIN {X 0,Y 587.375,Z 367.321,A -85,B 0,C 180,E1 -1622.743,E2 -1622.743} C_VEL
LIN {X 0,Y 587.362,Z 367.323,A -85,B 0,C 180,E1 -1625.493,E2 -1625.493} C_VEL
LIN {X 0,Y 587.37,Z 367.323,A -85,B 0,C 180,E1 -1628.255,E2 -1628.255} C_VEL
LIN {X 0,Y 587.352,Z 367.324,A -85,B 0,C 180,E1 -1631.134,E2 -1631.134} C_VEL
LIN {X 0,Y 587.368,Z 367.322,A -85,B 0,C 180,E1 -1634.26,E2 -1634.26} C_VEL
LIN {X 0,Y 587.351,Z 367.324,A -85,B 0,C 180,E1 -1637.406,E2 -1637.406} C_VEL
LIN {X 0,Y 587.31,Z 367.328,A -85,B 0,C 180,E1 -1638.314,E2 -1638.314} C_VEL
LIN {X 0,Y 586.669,Z 367.41,A -85,B 0,C 180,E1 -1638.886,E2 -1638.886} C_VEL
LIN {X 0,Y 583.846,Z 367.763,A -85,B 0,C 180,E1 -1639.814,E2 -1639.814} C_VEL
LIN {X 0,Y 581.435,Z 368.064,A -85,B 0,C 180,E1 -1640.561,E2 -1640.561} C_VEL
LIN {X 0,Y 580.381,Z 368.193,A -85,B 0,C 180,E1 -1641.138,E2 -1641.138} C_VEL
LIN {X 0,Y 580.285,Z 368.204,A -85,B 0,C 180,E1 -1641.333,E2 -1641.333} C_VEL
LIN {X 0,Y 580.283,Z 368.205,A -85,B 0,C 180,E1 -1643.558,E2 -1643.558} C_VEL
LIN {X 0,Y 580.283,Z 368.206,A -85,B 0,C 180,E1 -1645.849,E2 -1645.849} C_VEL
LIN {X 0,Y 580.303,Z 368.203,A -85,B 0,C 180,E1 -1648.185,E2 -1648.185} C_VEL
LIN {X 0,Y 580.289,Z 368.203,A -85,B 0,C 180,E1 -1650.694,E2 -1650.694} C_VEL
LIN {X 0,Y 580.288,Z 368.206,A -85,B 0,C 180,E1 -1653.313,E2 -1653.313} C_VEL
LIN {X 0,Y 580.249,Z 368.208,A -85,B 0,C 180,E1 -1655.756,E2 -1655.756} C_VEL
LIN {X 0,Y 580.288,Z 368.204,A -85,B 0,C 180,E1 -1658.146,E2 -1658.146} C_VEL
LIN {X 0,Y 580.3,Z 368.203,A -85,B 0,C 180,E1 -1660.843,E2 -1660.843} C_VEL
LIN {X 0,Y 580.276,Z 368.207,A -85,B 0,C 180,E1 -1663.658,E2 -1663.658} C_VEL
LIN {X 0,Y 580.279,Z 368.206,A -85,B 0,C 180,E1 -1666.609,E2 -1666.609} C_VEL
LIN {X 0,Y 580.304,Z 368.202,A -85,B 0,C 180,E1 -1669.156,E2 -1669.156} C_VEL
LIN {X 0,Y 580.294,Z 368.205,A -85,B 0,C 180,E1 -1671.927,E2 -1671.927} C_VEL
LIN {X 0,Y 580.258,Z 368.207,A -85,B 0,C 180,E1 -1674.452,E2 -1674.452} C_VEL
LIN {X 0,Y 580.295,Z 368.205,A -85,B 0,C 180,E1 -1676.975,E2 -1676.975} C_VEL
LIN {X 0,Y 580.292,Z 368.203,A -85,B 0,C 180,E1 -1679.424,E2 -1679.424} C_VEL
LIN {X 0,Y 580.296,Z 368.204,A -85,B 0,C 180,E1 -1682.142,E2 -1682.142} C_VEL
LIN {X 0,Y 580.311,Z 368.201,A -85,B 0,C 180,E1 -1684.92,E2 -1684.92} C_VEL
LIN {X 0,Y 580.278,Z 368.205,A -85,B 0,C 180,E1 -1687.947,E2 -1687.947} C_VEL
LIN {X 0,Y 580.305,Z 368.202,A -85,B 0,C 180,E1 -1690.913,E2 -1690.913} C_VEL
LIN {X 0,Y 580.278,Z 368.206,A -85,B 0,C 180,E1 -1693.824,E2 -1693.824} C_VEL
LIN {X 0,Y 580.333,Z 368.199,A -85,B 0,C 180,E1 -1695.982,E2 -1695.982} C_VEL
LIN {X 0,Y 580.227,Z 368.214,A -85,B 0,C 180,E1 -1698.116,E2 -1698.116} C_VEL
LIN {X 0,Y 580.19,Z 368.442,A -85,B 0,C 180,E1 -1698.865,E2 -1698.865} C_VEL
LIN {X 0,Y 580.192,Z 371.676,A -85,B 0,C 180,E1 -1701.641,E2 -1701.641} C_VEL
LIN {X 0,Y 580.11,Z 374.905,A -85,B 0,C 180,E1 -1704.437,E2 -1704.437} C_VEL
LIN {X 0,Y 580.089,Z 377.268,A -85,B 0,C 180,E1 -1706.526,E2 -1706.526} C_VEL
LIN {X 0,Y 580.048,Z 379.767,A -85,B 0,C 180,E1 -1708.61,E2 -1708.61} C_VEL
LIN {X 0,Y 580.037,Z 382.414,A -85,B 0,C 180,E1 -1710.693,E2 -1710.693} C_VEL
LIN {X 0,Y 580.063,Z 386.005,A -85,B 0,C 180,E1 -1713.472,E2 -1713.472} C_VEL
LIN {X 0,Y 580.048,Z 390.017,A -85,B 0,C 180,E1 -1716.52,E2 -1716.52} C_VEL
LIN {X 0,Y 579.994,Z 393.414,A -85,B 0,C 180,E1 -1719.062,E2 -1719.062} C_VEL
LIN {X 0,Y 580.021,Z 395.78,A -85,B 0,C 180,E1 -1720.752,E2 -1720.752} C_VEL
LIN {X 0,Y 580.769,Z 401.775,A -85,B 0,C 180,E1 -1720.894,E2 -1720.894} C_VEL
LIN {X 0,Y 580.701,Z 414.254,A -85,B 0,C 180,E1 -1721.253,E2 -1721.253} C_VEL
LIN {X 0,Y 580.578,Z 425.667,A -85,B 0,C 180,E1 -1721.709,E2 -1721.709} C_VEL
LIN {X 0,Y 580.459,Z 437.383,A -85,B 0,C 180,E1 -1722.32,E2 -1722.32} C_VEL
LIN {X 0,Y 580.417,Z 448.072,A -85,B 0,C 180,E1 -1723.032,E2 -1723.032} C_VEL
LIN {X 0,Y 580.295,Z 457.894,A -85,B 0,C 180,E1 -1723.837,E2 -1723.837} C_VEL
LIN {X 0,Y 580.248,Z 466.838,A -85,B 0,C 180,E1 -1724.734,E2 -1724.734} C_VEL
LIN {X 0,Y 580.182,Z 474.243,A -85,B 0,C 180,E1 -1725.634,E2 -1725.634} C_VEL
LIN {X 0,Y 580.137,Z 481.754,A -85,B 0,C 180,E1 -1726.766,E2 -1726.766} C_VEL
LIN {X 0,Y 580.093,Z 488.115,A -85,B 0,C 180,E1 -1727.994,E2 -1727.994} C_VEL
LIN {X 0,Y 580.092,Z 492.443,A -85,B 0,C 180,E1 -1729.092,E2 -1729.092} C_VEL
LIN {X 0,Y 580.068,Z 494.694,A -85,B 0,C 180,E1 -1729.829,E2 -1729.829} C_VEL
LIN {X 0,Y 580.038,Z 497.418,A -85,B 0,C 180,E1 -1731.098,E2 -1731.098} C_VEL
LIN {X 0,Y 580.029,Z 498.588,A -85,B 0,C 180,E1 -1732.06,E2 -1732.06} C_VEL
LIN {X 0,Y 580.043,Z 498.985,A -85,B 0,C 180,E1 -1732.95,E2 -1732.95} C_VEL
LIN {X 0,Y 580.023,Z 498.887,A -85,B 0,C 180,E1 -1733.567,E2 -1733.567} C_VEL
LIN {X 0,Y 580.039,Z 497.914,A -85,B 0,C 180,E1 -1734.669,E2 -1734.669} C_VEL
LIN {X 0,Y 580.04,Z 495.72,A -85,B 0,C 180,E1 -1735.859,E2 -1735.859} C_VEL
LIN {X 0,Y 580.061,Z 492.362,A -85,B 0,C 180,E1 -1737.021,E2 -1737.021} C_VEL
LIN {X 0,Y 580.12,Z 487.668,A -85,B 0,C 180,E1 -1738.193,E2 -1738.193} C_VEL
LIN {X 0,Y 580.128,Z 482.016,A -85,B 0,C 180,E1 -1739.279,E2 -1739.279} C_VEL
LIN {X 0,Y 580.224,Z 474.832,A -85,B 0,C 180,E1 -1740.376,E2 -1740.376} C_VEL
LIN {X 0,Y 580.25,Z 466.575,A -85,B 0,C 180,E1 -1741.385,E2 -1741.385} C_VEL
LIN {X 0,Y 580.33,Z 457.38,A -85,B 0,C 180,E1 -1742.299,E2 -1742.299} C_VEL
LIN {X 0,Y 580.419,Z 447.573,A -85,B 0,C 180,E1 -1743.096,E2 -1743.096} C_VEL
LIN {X 0,Y 580.503,Z 437.41,A -85,B 0,C 180,E1 -1743.768,E2 -1743.768} C_VEL
LIN {X 0,Y 580.624,Z 425.056,A -85,B 0,C 180,E1 -1744.408,E2 -1744.408} C_VEL
LIN {X 0,Y 580.68,Z 413.06,A -85,B 0,C 180,E1 -1744.878,E2 -1744.878} C_VEL
LIN {X 0,Y 580.769,Z 400.128,A -85,B 0,C 180,E1 -1745.236,E2 -1745.236} C_VEL
LIN {X 0,Y 580.064,Z 395.681,A -85,B 0,C 180,E1 -1745.345,E2 -1745.345} C_VEL
LIN {X 0,Y 580.021,Z 391.891,A -85,B 0,C 180,E1 -1748.164,E2 -1748.164} C_VEL
LIN {X 0,Y 580.036,Z 388.308,A -85,B 0,C 180,E1 -1750.863,E2 -1750.863} C_VEL
LIN {X 0,Y 580.063,Z 384.631,A -85,B 0,C 180,E1 -1753.675,E2 -1753.675} C_VEL
LIN {X 0,Y 580.072,Z 381.231,A -85,B 0,C 180,E1 -1756.323,E2 -1756.323} C_VEL
LIN {X 0,Y 580.077,Z 377.838,A -85,B 0,C 180,E1 -1759.138,E2 -1759.138} C_VEL
LIN {X 0,Y 580.106,Z 374.763,A -85,B 0,C 180,E1 -1761.947,E2 -1761.947} C_VEL
LIN {X 0,Y 580.144,Z 371.796,A -85,B 0,C 180,E1 -1764.445,E2 -1764.445} C_VEL
LIN {X 0,Y 580.175,Z 368.87,A -85,B 0,C 180,E1 -1766.968,E2 -1766.968} C_VEL
LIN {X 0,Y 580.207,Z 368.217,A -85,B 0,C 180,E1 -1767.98,E2 -1767.98} C_VEL
LIN {X 0,Y 580.278,Z 368.203,A -85,B 0,C 180,E1 -1770.227,E2 -1770.227} C_VEL
LIN {X 0,Y 580.275,Z 368.206,A -85,B 0,C 180,E1 -1772.598,E2 -1772.598} C_VEL
LIN {X 0,Y 580.302,Z 368.203,A -85,B 0,C 180,E1 -1775.268,E2 -1775.268} C_VEL
LIN {X 0,Y 580.273,Z 368.206,A -85,B 0,C 180,E1 -1777.947,E2 -1777.947} C_VEL
LIN {X 0,Y 580.316,Z 368.199,A -85,B 0,C 180,E1 -1780.914,E2 -1780.914} C_VEL
LIN {X 0,Y 580.263,Z 368.205,A -85,B 0,C 180,E1 -1783.825,E2 -1783.825} C_VEL
LIN {X 0,Y 580.317,Z 368.202,A -85,B 0,C 180,E1 -1785.983,E2 -1785.983} C_VEL
LIN {X 0,Y 580.33,Z 368.198,A -85,B 0,C 180,E1 -1788.827,E2 -1788.827} C_VEL
LIN {X 0,Y 580.316,Z 368.199,A -85,B 0,C 180,E1 -1791.644,E2 -1791.644} C_VEL
LIN {X 0,Y 580.322,Z 368.198,A -85,B 0,C 180,E1 -1794.44,E2 -1794.44} C_VEL
LIN {X 0,Y 580.33,Z 368.197,A -85,B 0,C 180,E1 -1797.223,E2 -1797.223} C_VEL
LIN {X 0,Y 580.327,Z 368.197,A -85,B 0,C 180,E1 -1800,E2 -1800} C_VEL
LIN {X 0,Y 580.333,Z 368.196,A -85,B 0,C 180,E1 -1802.777,E2 -1802.777} C_VEL
LIN {X 0,Y 580.31,Z 368.199,A -85,B 0,C 180,E1 -1805.56,E2 -1805.56} C_VEL
LIN {X 0,Y 580.314,Z 368.199,A -85,B 0,C 180,E1 -1808.356,E2 -1808.356} C_VEL
LIN {X 0,Y 580.312,Z 368.199,A -85,B 0,C 180,E1 -1811.209,E2 -1811.209} C_VEL
LIN {X 0,Y 580.294,Z 368.205,A -85,B 0,C 180,E1 -1814.34,E2 -1814.34} C_VEL
LIN {X 0,Y 580.293,Z 368.205,A -85,B 0,C 180,E1 -1816.916,E2 -1816.916} C_VEL
LIN {X 0,Y 580.294,Z 368.204,A -85,B 0,C 180,E1 -1819.823,E2 -1819.823} C_VEL
LIN {X 0,Y 580.333,Z 368.197,A -85,B 0,C 180,E1 -1822.801,E2 -1822.801} C_VEL
LIN {X 0,Y 580.276,Z 368.204,A -85,B 0,C 180,E1 -1825.85,E2 -1825.85} C_VEL
LIN {X 0,Y 580.288,Z 368.203,A -85,B 0,C 180,E1 -1828.186,E2 -1828.186} C_VEL
LIN {X 0,Y 580.276,Z 368.206,A -85,B 0,C 180,E1 -1830.698,E2 -1830.698} C_VEL
LIN {X 0,Y 580.288,Z 368.205,A -85,B 0,C 180,E1 -1833.318,E2 -1833.318} C_VEL
LIN {X 0,Y 580.312,Z 368.202,A -85,B 0,C 180,E1 -1835.769,E2 -1835.769} C_VEL
LIN {X 0,Y 580.272,Z 368.204,A -85,B 0,C 180,E1 -1838.148,E2 -1838.148} C_VEL
LIN {X 0,Y 580.307,Z 368.2,A -85,B 0,C 180,E1 -1840.843,E2 -1840.843} C_VEL
LIN {X 0,Y 580.266,Z 368.207,A -85,B 0,C 180,E1 -1843.659,E2 -1843.659} C_VEL
LIN {X 0,Y 580.272,Z 368.208,A -85,B 0,C 180,E1 -1846.61,E2 -1846.61} C_VEL
LIN {X 0,Y 580.31,Z 368.202,A -85,B 0,C 180,E1 -1849.16,E2 -1849.16} C_VEL
LIN {X 0,Y 580.28,Z 368.206,A -85,B 0,C 180,E1 -1851.929,E2 -1851.929} C_VEL
LIN {X 0,Y 580.341,Z 368.336,A -85,B 0,C 180,E1 -1853.509,E2 -1853.509} C_VEL
LIN {X 0,Y 580.721,Z 371.276,A -85,B 0,C 180,E1 -1854.488,E2 -1854.488} C_VEL
LIN {X 0,Y 580.674,Z 379.22,A -85,B 0,C 180,E1 -1857.002,E2 -1857.002} C_VEL
LIN {X 0,Y 580.547,Z 387.163,A -85,B 0,C 180,E1 -1859.442,E2 -1859.442} C_VEL
LIN {X 0,Y 580.519,Z 396.024,A -85,B 0,C 180,E1 -1862.101,E2 -1862.101} C_VEL
LIN {X 0,Y 580.429,Z 405.697,A -85,B 0,C 180,E1 -1864.928,E2 -1864.928} C_VEL
LIN {X 0,Y 580.371,Z 414.964,A -85,B 0,C 180,E1 -1867.578,E2 -1867.578} C_VEL
LIN {X 0,Y 580.312,Z 424.231,A -85,B 0,C 180,E1 -1870.18,E2 -1870.18} C_VEL
LIN {X 0,Y 580.227,Z 434.872,A -85,B 0,C 180,E1 -1873.115,E2 -1873.115} C_VEL
LIN {X 0,Y 580.185,Z 445.413,A -85,B 0,C 180,E1 -1875.981,E2 -1875.981} C_VEL
LIN {X 0,Y 580.141,Z 451.578,A -85,B 0,C 180,E1 -1877.64,E2 -1877.64} C_VEL
LIN {X 0,Y 580.805,Z 457.313,A -85,B 0,C 180,E1 -1877.754,E2 -1877.754} C_VEL
LIN {X 0,Y 580.74,Z 470.551,A -85,B 0,C 180,E1 -1878.085,E2 -1878.085} C_VEL
LIN {X 0,Y 580.616,Z 482.357,A -85,B 0,C 180,E1 -1878.516,E2 -1878.516} C_VEL
LIN {X 0,Y 580.5,Z 494.237,A -85,B 0,C 180,E1 -1879.097,E2 -1879.097} C_VEL
LIN {X 0,Y 580.457,Z 505.5,A -85,B 0,C 180,E1 -1879.802,E2 -1879.802} C_VEL
LIN {X 0,Y 580.352,Z 515.665,A -85,B 0,C 180,E1 -1880.592,E2 -1880.592} C_VEL
LIN {X 0,Y 580.278,Z 524.801,A -85,B 0,C 180,E1 -1881.469,E2 -1881.469} C_VEL
LIN {X 0,Y 580.198,Z 533.702,A -85,B 0,C 180,E1 -1882.519,E2 -1882.519} C_VEL
LIN {X 0,Y 580.119,Z 540.47,A -85,B 0,C 180,E1 -1883.505,E2 -1883.505} C_VEL
LIN {X 0,Y 580.139,Z 545.688,A -85,B 0,C 180,E1 -1884.44,E2 -1884.44} C_VEL
LIN {X 0,Y 580.108,Z 550.377,A -85,B 0,C 180,E1 -1885.485,E2 -1885.485} C_VEL
LIN {X 0,Y 580.122,Z 553.961,A -85,B 0,C 180,E1 -1886.529,E2 -1886.529} C_VEL
LIN {X 0,Y 580.043,Z 555.812,A -85,B 0,C 180,E1 -1887.223,E2 -1887.223} C_VEL
LIN {X 0,Y 580.04,Z 557.203,A -85,B 0,C 180,E1 -1887.918,E2 -1887.918} C_VEL
LIN {X 0,Y 580.04,Z 558.785,A -85,B 0,C 180,E1 -1889.307,E2 -1889.307} C_VEL
LIN {X 0,Y 580.037,Z 559,A -85,B 0,C 180,E1 -1890.001,E2 -1890.001} C_VEL
LIN {X 0,Y 580.047,Z 558.183,A -85,B 0,C 180,E1 -1891.39,E2 -1891.39} C_VEL
LIN {X 0,Y 580.04,Z 557.2,A -85,B 0,C 180,E1 -1892.084,E2 -1892.084} C_VEL
LIN {X 0,Y 580.043,Z 555.806,A -85,B 0,C 180,E1 -1892.779,E2 -1892.779} C_VEL
LIN {X 0,Y 580.11,Z 552.892,A -85,B 0,C 180,E1 -1893.822,E2 -1893.822} C_VEL
LIN {X 0,Y 580.053,Z 548.945,A -85,B 0,C 180,E1 -1894.866,E2 -1894.866} C_VEL
LIN {X 0,Y 580.139,Z 542.87,A -85,B 0,C 180,E1 -1896.086,E2 -1896.086} C_VEL
LIN {X 0,Y 580.185,Z 536.228,A -85,B 0,C 180,E1 -1897.134,E2 -1897.134} C_VEL
LIN {X 0,Y 580.251,Z 527.98,A -85,B 0,C 180,E1 -1898.183,E2 -1898.183} C_VEL
LIN {X 0,Y 580.309,Z 519.524,A -85,B 0,C 180,E1 -1899.06,E2 -1899.06} C_VEL
LIN {X 0,Y 580.424,Z 509.078,A -85,B 0,C 180,E1 -1899.937,E2 -1899.937} C_VEL
LIN {X 0,Y 580.5,Z 498.74,A -85,B 0,C 180,E1 -1900.641,E2 -1900.641} C_VEL
LIN {X 0,Y 580.566,Z 487.571,A -85,B 0,C 180,E1 -1901.249,E2 -1901.249} C_VEL
LIN {X 0,Y 580.667,Z 475.734,A -85,B 0,C 180,E1 -1901.742,E2 -1901.742} C_VEL
LIN {X 0,Y 580.776,Z 462.305,A -85,B 0,C 180,E1 -1902.138,E2 -1902.138} C_VEL
LIN {X 0,Y 580.598,Z 454.43,A -85,B 0,C 180,E1 -1902.306,E2 -1902.306} C_VEL
LIN {X 0,Y 580.129,Z 451.526,A -85,B 0,C 180,E1 -1902.374,E2 -1902.374} C_VEL
LIN {X 0,Y 580.219,Z 441.432,A -85,B 0,C 180,E1 -1905.096,E2 -1905.096} C_VEL
LIN {X 0,Y 580.255,Z 430.841,A -85,B 0,C 180,E1 -1907.991,E2 -1907.991} C_VEL
LIN {X 0,Y 580.337,Z 420.488,A -85,B 0,C 180,E1 -1910.866,E2 -1910.866} C_VEL
LIN {X 0,Y 580.385,Z 410.983,A -85,B 0,C 180,E1 -1913.554,E2 -1913.554} C_VEL
LIN {X 0,Y 580.484,Z 401.22,A -85,B 0,C 180,E1 -1916.372,E2 -1916.372} C_VEL
LIN {X 0,Y 580.533,Z 391.162,A -85,B 0,C 180,E1 -1919.35,E2 -1919.35} C_VEL
LIN {X 0,Y 580.672,Z 381.857,A -85,B 0,C 180,E1 -1922.178,E2 -1922.178} C_VEL
LIN {X 0,Y 580.716,Z 373.914,A -85,B 0,C 180,E1 -1924.668,E2 -1924.668} C_VEL
LIN {X 0,Y 580.67,Z 370.351,A -85,B 0,C 180,E1 -1925.814,E2 -1925.814} C_VEL
LIN {X 0,Y 580.309,Z 368.202,A -85,B 0,C 180,E1 -1926.591,E2 -1926.591} C_VEL
LIN {X 0,Y 580.298,Z 368.205,A -85,B 0,C 180,E1 -1929.185,E2 -1929.185} C_VEL
LIN {X 0,Y 580.286,Z 368.204,A -85,B 0,C 180,E1 -1931.769,E2 -1931.769} C_VEL
LIN {X 0,Y 580.253,Z 368.21,A -85,B 0,C 180,E1 -1934.628,E2 -1934.628} C_VEL
LIN {X 0,Y 580.291,Z 368.206,A -85,B 0,C 180,E1 -1937.628,E2 -1937.628} C_VEL
LIN {X 0,Y 580.287,Z 368.204,A -85,B 0,C 180,E1 -1940.066,E2 -1940.066} C_VEL
LIN {X 0,Y 580.303,Z 368.202,A -85,B 0,C 180,E1 -1943.066,E2 -1943.066} C_VEL
LIN {X 0,Y 580.305,Z 368.202,A -85,B 0,C 180,E1 -1946.144,E2 -1946.144} C_VEL
LIN {X 0,Y 580.28,Z 368.205,A -85,B 0,C 180,E1 -1948.615,E2 -1948.615} C_VEL
LIN {X 0,Y 580.296,Z 368.205,A -85,B 0,C 180,E1 -1951.024,E2 -1951.024} C_VEL
LIN {X 0,Y 580.295,Z 368.202,A -85,B 0,C 180,E1 -1953.666,E2 -1953.666} C_VEL
LIN {X 0,Y 580.3,Z 368.202,A -85,B 0,C 180,E1 -1955.684,E2 -1955.684} C_VEL
LIN {X 0,Y 580.273,Z 368.206,A -85,B 0,C 180,E1 -1957.947,E2 -1957.947} C_VEL
LIN {X 0,Y 580.323,Z 368.199,A -85,B 0,C 180,E1 -1960.914,E2 -1960.914} C_VEL
LIN {X 0,Y 580.28,Z 368.205,A -85,B 0,C 180,E1 -1963.825,E2 -1963.825} C_VEL
LIN {X 0,Y 580.328,Z 368.199,A -85,B 0,C 180,E1 -1965.983,E2 -1965.983} C_VEL
LIN {X 0,Y 580.309,Z 368.202,A -85,B 0,C 180,E1 -1968.827,E2 -1968.827} C_VEL
LIN {X 0,Y 580.335,Z 368.199,A -85,B 0,C 180,E1 -1971.644,E2 -1971.644} C_VEL
LIN {X 0,Y 580.324,Z 368.199,A -85,B 0,C 180,E1 -1974.44,E2 -1974.44} C_VEL
LIN {X 0,Y 580.337,Z 368.198,A -85,B 0,C 180,E1 -1977.223,E2 -1977.223} C_VEL
LIN {X 0,Y 580.354,Z 368.197,A -85,B 0,C 180,E1 -1980,E2 -1980} C_VEL
LIN {X 0,Y 580.342,Z 368.197,A -85,B 0,C 180,E1 -1982.776,E2 -1982.776} C_VEL
LIN {X 0,Y 580.327,Z 368.199,A -85,B 0,C 180,E1 -1985.56,E2 -1985.56} C_VEL
LIN {X 0,Y 580.335,Z 368.2,A -85,B 0,C 180,E1 -1988.356,E2 -1988.356} C_VEL
LIN {X 0,Y 580.304,Z 368.202,A -85,B 0,C 180,E1 -1991.191,E2 -1991.191} C_VEL
LIN {X 0,Y 580.327,Z 368.199,A -85,B 0,C 180,E1 -1994.017,E2 -1994.017} C_VEL
LIN {X 0,Y 580.316,Z 368.201,A -85,B 0,C 180,E1 -1996.914,E2 -1996.914} C_VEL
LIN {X 0,Y 580.289,Z 368.206,A -85,B 0,C 180,E1 -1999.823,E2 -1999.823} C_VEL
LIN {X 0,Y 580.285,Z 368.204,A -85,B 0,C 180,E1 -2001.333,E2 -2001.333} C_VEL
LIN {X 0,Y 579.587,Z 368.293,A -85,B 0,C 180,E1 -2001.912,E2 -2001.912} C_VEL
LIN {X 0,Y 576.711,Z 368.651,A -85,B 0,C 180,E1 -2002.852,E2 -2002.852} C_VEL
LIN {X 0,Y 574.318,Z 368.948,A -85,B 0,C 180,E1 -2003.608,E2 -2003.608} C_VEL
LIN {X 0,Y 573.32,Z 369.072,A -85,B 0,C 180,E1 -2004.192,E2 -2004.192} C_VEL
LIN {X 0,Y 573.254,Z 369.079,A -85,B 0,C 180,E1 -2004.39,E2 -2004.39} C_VEL
LIN {X 0,Y 573.254,Z 369.082,A -85,B 0,C 180,E1 -2006.976,E2 -2006.976} C_VEL
LIN {X 0,Y 573.25,Z 369.081,A -85,B 0,C 180,E1 -2009.488,E2 -2009.488} C_VEL
LIN {X 0,Y 573.258,Z 369.079,A -85,B 0,C 180,E1 -2012.645,E2 -2012.645} C_VEL
LIN {X 0,Y 573.211,Z 369.087,A -85,B 0,C 180,E1 -2015.188,E2 -2015.188} C_VEL
LIN {X 0,Y 573.237,Z 369.082,A -85,B 0,C 180,E1 -2017.808,E2 -2017.808} C_VEL
LIN {X 0,Y 573.249,Z 369.083,A -85,B 0,C 180,E1 -2020.525,E2 -2020.525} C_VEL
LIN {X 0,Y 573.24,Z 369.083,A -85,B 0,C 180,E1 -2023.359,E2 -2023.359} C_VEL
LIN {X 0,Y 573.242,Z 369.083,A -85,B 0,C 180,E1 -2026.64,E2 -2026.64} C_VEL
LIN {X 0,Y 573.249,Z 369.081,A -85,B 0,C 180,E1 -2029.474,E2 -2029.474} C_VEL
LIN {X 0,Y 573.24,Z 369.082,A -85,B 0,C 180,E1 -2032.192,E2 -2032.192} C_VEL
LIN {X 0,Y 573.241,Z 369.082,A -85,B 0,C 180,E1 -2035.228,E2 -2035.228} C_VEL
LIN {X 0,Y 573.256,Z 369.08,A -85,B 0,C 180,E1 -2037.771,E2 -2037.771} C_VEL
LIN {X 0,Y 573.266,Z 369.078,A -85,B 0,C 180,E1 -2040.633,E2 -2040.633} C_VEL
LIN {X 0,Y 573.241,Z 369.082,A -85,B 0,C 180,E1 -2043.507,E2 -2043.507} C_VEL
LIN {X 0,Y 573.236,Z 369.082,A -85,B 0,C 180,E1 -2046.134,E2 -2046.134} C_VEL
LIN {X 0,Y 573.256,Z 369.08,A -85,B 0,C 180,E1 -2049.173,E2 -2049.173} C_VEL
LIN {X 0,Y 573.227,Z 369.084,A -85,B 0,C 180,E1 -2051.41,E2 -2051.41} C_VEL
LIN {X 0,Y 573.25,Z 369.082,A -85,B 0,C 180,E1 -2053.621,E2 -2053.621} C_VEL
LIN {X 0,Y 573.28,Z 369.079,A -85,B 0,C 180,E1 -2055.806,E2 -2055.806} C_VEL
LIN {X 0,Y 573.149,Z 369.095,A -85,B 0,C 180,E1 -2058.684,E2 -2058.684} C_VEL
LIN {X 0,Y 573.129,Z 372.185,A -85,B 0,C 180,E1 -2061.537,E2 -2061.537} C_VEL
LIN {X 0,Y 573.043,Z 375.43,A -85,B 0,C 180,E1 -2064.368,E2 -2064.368} C_VEL
LIN {X 0,Y 573.022,Z 377.792,A -85,B 0,C 180,E1 -2066.483,E2 -2066.483} C_VEL
LIN {X 0,Y 572.973,Z 381.033,A -85,B 0,C 180,E1 -2069.296,E2 -2069.296} C_VEL
LIN {X 0,Y 572.958,Z 384.58,A -85,B 0,C 180,E1 -2072.107,E2 -2072.107} C_VEL
LIN {X 0,Y 572.979,Z 387.295,A -85,B 0,C 180,E1 -2074.219,E2 -2074.219} C_VEL
LIN {X 0,Y 572.951,Z 390.982,A -85,B 0,C 180,E1 -2077.044,E2 -2077.044} C_VEL
LIN {X 0,Y 572.948,Z 394.743,A -85,B 0,C 180,E1 -2079.887,E2 -2079.887} C_VEL
LIN {X 0,Y 572.931,Z 395.667,A -85,B 0,C 180,E1 -2080.579,E2 -2080.579} C_VEL
LIN {X 0,Y 573.82,Z 402.252,A -85,B 0,C 180,E1 -2080.756,E2 -2080.756} C_VEL
LIN {X 0,Y 573.755,Z 414.527,A -85,B 0,C 180,E1 -2081.118,E2 -2081.118} C_VEL
LIN {X 0,Y 573.609,Z 426.494,A -85,B 0,C 180,E1 -2081.607,E2 -2081.607} C_VEL
LIN {X 0,Y 573.481,Z 437.621,A -85,B 0,C 180,E1 -2082.203,E2 -2082.203} C_VEL
LIN {X 0,Y 573.408,Z 448.275,A -85,B 0,C 180,E1 -2082.924,E2 -2082.924} C_VEL
LIN {X 0,Y 573.246,Z 459.06,A -85,B 0,C 180,E1 -2083.83,E2 -2083.83} C_VEL
LIN {X 0,Y 573.175,Z 467.996,A -85,B 0,C 180,E1 -2084.762,E2 -2084.762} C_VEL
LIN {X 0,Y 573.115,Z 476.292,A -85,B 0,C 180,E1 -2085.832,E2 -2085.832} C_VEL
LIN {X 0,Y 573.072,Z 483.233,A -85,B 0,C 180,E1 -2086.947,E2 -2086.947} C_VEL
LIN {X 0,Y 573.005,Z 487.765,A -85,B 0,C 180,E1 -2087.854,E2 -2087.854} C_VEL
LIN {X 0,Y 573.007,Z 491.908,A -85,B 0,C 180,E1 -2088.89,E2 -2088.89} C_VEL
LIN {X 0,Y 572.982,Z 495.441,A -85,B 0,C 180,E1 -2090.085,E2 -2090.085} C_VEL
LIN {X 0,Y 572.96,Z 497.64,A -85,B 0,C 180,E1 -2091.215,E2 -2091.215} C_VEL
LIN {X 0,Y 572.934,Z 498.789,A -85,B 0,C 180,E1 -2092.348,E2 -2092.348} C_VEL
LIN {X 0,Y 572.932,Z 498.992,A -85,B 0,C 180,E1 -2093.11,E2 -2093.11} C_VEL
LIN {X 0,Y 572.923,Z 498.699,A -85,B 0,C 180,E1 -2093.877,E2 -2093.877} C_VEL
LIN {X 0,Y 572.933,Z 497.748,A -85,B 0,C 180,E1 -2094.805,E2 -2094.805} C_VEL
LIN {X 0,Y 572.985,Z 494.945,A -85,B 0,C 180,E1 -2096.201,E2 -2096.201} C_VEL
LIN {X 0,Y 573.006,Z 491.269,A -85,B 0,C 180,E1 -2097.381,E2 -2097.381} C_VEL
LIN {X 0,Y 573.021,Z 486.2,A -85,B 0,C 180,E1 -2098.574,E2 -2098.574} C_VEL
LIN {X 0,Y 573.083,Z 479.395,A -85,B 0,C 180,E1 -2099.79,E2 -2099.79} C_VEL
LIN {X 0,Y 573.155,Z 471.776,A -85,B 0,C 180,E1 -2100.87,E2 -2100.87} C_VEL
LIN {X 0,Y 573.234,Z 463.577,A -85,B 0,C 180,E1 -2101.814,E2 -2101.814} C_VEL
LIN {X 0,Y 573.337,Z 453.621,A -85,B 0,C 180,E1 -2102.742,E2 -2102.742} C_VEL
LIN {X 0,Y 573.413,Z 442.958,A -85,B 0,C 180,E1 -2103.546,E2 -2103.546} C_VEL
LIN {X 0,Y 573.569,Z 431.098,A -85,B 0,C 180,E1 -2104.253,E2 -2104.253} C_VEL
LIN {X 0,Y 573.695,Z 418.213,A -85,B 0,C 180,E1 -2104.837,E2 -2104.837} C_VEL
LIN {X 0,Y 573.804,Z 405.632,A -85,B 0,C 180,E1 -2105.251,E2 -2105.251} C_VEL
LIN {X 0,Y 573.653,Z 400.002,A -85,B 0,C 180,E1 -2105.392,E2 -2105.392} C_VEL
LIN {X 0,Y 572.957,Z 395.68,A -85,B 0,C 180,E1 -2105.5,E2 -2105.5} C_VEL
LIN {X 0,Y 572.936,Z 392,A -85,B 0,C 180,E1 -2108.273,E2 -2108.273} C_VEL
LIN {X 0,Y 572.971,Z 389.017,A -85,B 0,C 180,E1 -2110.546,E2 -2110.546} C_VEL
LIN {X 0,Y 572.975,Z 385.349,A -85,B 0,C 180,E1 -2113.381,E2 -2113.381} C_VEL
LIN {X 0,Y 573.002,Z 382.468,A -85,B 0,C 180,E1 -2115.644,E2 -2115.644} C_VEL
LIN {X 0,Y 573.011,Z 379.137,A -85,B 0,C 180,E1 -2118.524,E2 -2118.524} C_VEL
LIN {X 0,Y 573.012,Z 376.146,A -85,B 0,C 180,E1 -2121.28,E2 -2121.28} C_VEL
LIN {X 0,Y 573.069,Z 372.864,A -85,B 0,C 180,E1 -2124.034,E2 -2124.034} C_VEL
LIN {X 0,Y 573.09,Z 370.061,A -85,B 0,C 180,E1 -2126.506,E2 -2126.506} C_VEL
LIN {X 0,Y 573.089,Z 369.103,A -85,B 0,C 180,E1 -2127.344,E2 -2127.344} C_VEL
LIN {X 0,Y 573.239,Z 369.083,A -85,B 0,C 180,E1 -2129.823,E2 -2129.823} C_VEL
LIN {X 0,Y 573.272,Z 369.079,A -85,B 0,C 180,E1 -2132.234,E2 -2132.234} C_VEL
LIN {X 0,Y 573.249,Z 369.083,A -85,B 0,C 180,E1 -2135.12,E2 -2135.12} C_VEL
LIN {X 0,Y 573.249,Z 369.082,A -85,B 0,C 180,E1 -2137.663,E2 -2137.663} C_VEL
LIN {X 0,Y 573.259,Z 369.079,A -85,B 0,C 180,E1 -2140.727,E2 -2140.727} C_VEL
LIN {X 0,Y 573.239,Z 369.08,A -85,B 0,C 180,E1 -2143.621,E2 -2143.621} C_VEL
LIN {X 0,Y 573.264,Z 369.08,A -85,B 0,C 180,E1 -2145.807,E2 -2145.807} C_VEL
LIN {X 0,Y 573.262,Z 369.08,A -85,B 0,C 180,E1 -2148.734,E2 -2148.734} C_VEL
LIN {X 0,Y 573.288,Z 369.076,A -85,B 0,C 180,E1 -2151.541,E2 -2151.541} C_VEL
LIN {X 0,Y 573.289,Z 369.074,A -85,B 0,C 180,E1 -2154.372,E2 -2154.372} C_VEL
LIN {X 0,Y 573.305,Z 369.074,A -85,B 0,C 180,E1 -2157.892,E2 -2157.892} C_VEL
LIN {X 0,Y 573.324,Z 369.073,A -85,B 0,C 180,E1 -2160.702,E2 -2160.702} C_VEL
LIN {X 0,Y 573.233,Z 369.084,A -85,B 0,C 180,E1 -2163.515,E2 -2163.515} C_VEL
LIN {X 0,Y 573.276,Z 369.075,A -85,B 0,C 180,E1 -2165.628,E2 -2165.628} C_VEL
LIN {X 0,Y 573.27,Z 369.077,A -85,B 0,C 180,E1 -2168.46,E2 -2168.46} C_VEL
LIN {X 0,Y 573.278,Z 369.076,A -85,B 0,C 180,E1 -2171.312,E2 -2171.312} C_VEL
LIN {X 0,Y 573.26,Z 369.08,A -85,B 0,C 180,E1 -2174.425,E2 -2174.425} C_VEL
LIN {X 0,Y 573.24,Z 369.083,A -85,B 0,C 180,E1 -2177.112,E2 -2177.112} C_VEL
LIN {X 0,Y 573.242,Z 369.08,A -85,B 0,C 180,E1 -2180.077,E2 -2180.077} C_VEL
LIN {X 0,Y 573.275,Z 369.076,A -85,B 0,C 180,E1 -2183.16,E2 -2183.16} C_VEL
LIN {X 0,Y 573.27,Z 369.078,A -85,B 0,C 180,E1 -2186.19,E2 -2186.19} C_VEL
LIN {X 0,Y 573.226,Z 369.082,A -85,B 0,C 180,E1 -2188.565,E2 -2188.565} C_VEL
LIN {X 0,Y 573.22,Z 369.083,A -85,B 0,C 180,E1 -2190.994,E2 -2190.994} C_VEL
LIN {X 0,Y 573.245,Z 369.081,A -85,B 0,C 180,E1 -2193.525,E2 -2193.525} C_VEL
LIN {X 0,Y 573.247,Z 369.082,A -85,B 0,C 180,E1 -2196.049,E2 -2196.049} C_VEL
LIN {X 0,Y 573.228,Z 369.085,A -85,B 0,C 180,E1 -2198.703,E2 -2198.703} C_VEL
LIN {X 0,Y 573.253,Z 369.081,A -85,B 0,C 180,E1 -2201.599,E2 -2201.599} C_VEL
LIN {X 0,Y 573.212,Z 369.085,A -85,B 0,C 180,E1 -2204.677,E2 -2204.677} C_VEL
LIN {X 0,Y 573.231,Z 369.082,A -85,B 0,C 180,E1 -2207.36,E2 -2207.36} C_VEL
LIN {X 0,Y 573.263,Z 369.081,A -85,B 0,C 180,E1 -2209.479,E2 -2209.479} C_VEL
LIN {X 0,Y 573.227,Z 369.086,A -85,B 0,C 180,E1 -2212.194,E2 -2212.194} C_VEL
LIN {X 0,Y 573.31,Z 369.292,A -85,B 0,C 180,E1 -2213.304,E2 -2213.304} C_VEL
LIN {X 0,Y 573.779,Z 372.6,A -85,B 0,C 180,E1 -2214.425,E2 -2214.425} C_VEL
LIN {X 0,Y 573.706,Z 380.544,A -85,B 0,C 180,E1 -2216.969,E2 -2216.969} C_VEL
LIN {X 0,Y 573.58,Z 388.529,A -85,B 0,C 180,E1 -2219.452,E2 -2219.452} C_VEL
LIN {X 0,Y 573.494,Z 397.754,A -85,B 0,C 180,E1 -2222.248,E2 -2222.248} C_VEL
LIN {X 0,Y 573.425,Z 407.365,A -85,B 0,C 180,E1 -2225.089,E2 -2225.089} C_VEL
LIN {X 0,Y 573.348,Z 417.612,A -85,B 0,C 180,E1 -2228.048,E2 -2228.048} C_VEL
LIN {X 0,Y 573.224,Z 428.336,A -85,B 0,C 180,E1 -2231.079,E2 -2231.079} C_VEL
LIN {X 0,Y 573.164,Z 438.794,A -85,B 0,C 180,E1 -2233.987,E2 -2233.987} C_VEL
LIN {X 0,Y 573.097,Z 449.385,A -85,B 0,C 180,E1 -2236.889,E2 -2236.889} C_VEL
LIN {X 0,Y 573.084,Z 451.536,A -85,B 0,C 180,E1 -2237.474,E2 -2237.474} C_VEL
LIN {X 0,Y 573.874,Z 457.313,A -85,B 0,C 180,E1 -2237.604,E2 -2237.604} C_VEL
LIN {X 0,Y 573.79,Z 470.552,A -85,B 0,C 180,E1 -2237.939,E2 -2237.939} C_VEL
LIN {X 0,Y 573.652,Z 482.786,A -85,B 0,C 180,E1 -2238.394,E2 -2238.394} C_VEL
LIN {X 0,Y 573.523,Z 494.457,A -85,B 0,C 180,E1 -2238.976,E2 -2238.976} C_VEL
LIN {X 0,Y 573.451,Z 505.5,A -85,B 0,C 180,E1 -2239.676,E2 -2239.676} C_VEL
LIN {X 0,Y 573.307,Z 515.665,A -85,B 0,C 180,E1 -2240.476,E2 -2240.476} C_VEL
LIN {X 0,Y 573.214,Z 524.801,A -85,B 0,C 180,E1 -2241.363,E2 -2241.363} C_VEL
LIN {X 0,Y 573.141,Z 533.702,A -85,B 0,C 180,E1 -2242.427,E2 -2242.427} C_VEL
LIN {X 0,Y 573.05,Z 540.411,A -85,B 0,C 180,E1 -2243.416,E2 -2243.416} C_VEL
LIN {X 0,Y 573.07,Z 545.688,A -85,B 0,C 180,E1 -2244.371,E2 -2244.371} C_VEL
LIN {X 0,Y 573.028,Z 550.377,A -85,B 0,C 180,E1 -2245.429,E2 -2245.429} C_VEL
LIN {X 0,Y 573.022,Z 553.961,A -85,B 0,C 180,E1 -2246.486,E2 -2246.486} C_VEL
LIN {X 0,Y 572.959,Z 555.812,A -85,B 0,C 180,E1 -2247.189,E2 -2247.189} C_VEL
LIN {X 0,Y 572.939,Z 557.203,A -85,B 0,C 180,E1 -2247.892,E2 -2247.892} C_VEL
LIN {X 0,Y 572.94,Z 558.785,A -85,B 0,C 180,E1 -2249.299,E2 -2249.299} C_VEL
LIN {X 0,Y 572.938,Z 559,A -85,B 0,C 180,E1 -2250.001,E2 -2250.001} C_VEL
LIN {X 0,Y 572.946,Z 558.184,A -85,B 0,C 180,E1 -2251.407,E2 -2251.407} C_VEL
LIN {X 0,Y 572.94,Z 557.199,A -85,B 0,C 180,E1 -2252.11,E2 -2252.11} C_VEL
LIN {X 0,Y 572.959,Z 555.807,A -85,B 0,C 180,E1 -2252.814,E2 -2252.814} C_VEL
LIN {X 0,Y 573.015,Z 552.892,A -85,B 0,C 180,E1 -2253.869,E2 -2253.869} C_VEL
LIN {X 0,Y 572.963,Z 548.944,A -85,B 0,C 180,E1 -2254.927,E2 -2254.927} C_VEL
LIN {X 0,Y 573.065,Z 542.87,A -85,B 0,C 180,E1 -2256.161,E2 -2256.161} C_VEL
LIN {X 0,Y 573.121,Z 536.228,A -85,B 0,C 180,E1 -2257.222,E2 -2257.222} C_VEL
LIN {X 0,Y 573.199,Z 527.98,A -85,B 0,C 180,E1 -2258.284,E2 -2258.284} C_VEL
LIN {X 0,Y 573.288,Z 519.525,A -85,B 0,C 180,E1 -2259.171,E2 -2259.171} C_VEL
LIN {X 0,Y 573.418,Z 509.079,A -85,B 0,C 180,E1 -2260.06,E2 -2260.06} C_VEL
LIN {X 0,Y 573.523,Z 497.515,A -85,B 0,C 180,E1 -2260.848,E2 -2260.848} C_VEL
LIN {X 0,Y 573.613,Z 485.854,A -85,B 0,C 180,E1 -2261.467,E2 -2261.467} C_VEL
LIN {X 0,Y 573.751,Z 473.143,A -85,B 0,C 180,E1 -2261.975,E2 -2261.975} C_VEL
LIN {X 0,Y 573.869,Z 460.476,A -85,B 0,C 180,E1 -2262.332,E2 -2262.332} C_VEL
LIN {X 0,Y 573.711,Z 455.603,A -85,B 0,C 180,E1 -2262.433,E2 -2262.433} C_VEL
LIN {X 0,Y 573.086,Z 451.526,A -85,B 0,C 180,E1 -2262.529,E2 -2262.529} C_VEL
LIN {X 0,Y 573.159,Z 441.432,A -85,B 0,C 180,E1 -2265.287,E2 -2265.287} C_VEL
LIN {X 0,Y 573.217,Z 430.841,A -85,B 0,C 180,E1 -2268.22,E2 -2268.22} C_VEL
LIN {X 0,Y 573.303,Z 421.573,A -85,B 0,C 180,E1 -2270.825,E2 -2270.825} C_VEL
LIN {X 0,Y 573.356,Z 412.308,A -85,B 0,C 180,E1 -2273.477,E2 -2273.477} C_VEL
LIN {X 0,Y 573.457,Z 403.039,A -85,B 0,C 180,E1 -2276.181,E2 -2276.181} C_VEL
LIN {X 0,Y 573.496,Z 393.772,A -85,B 0,C 180,E1 -2278.952,E2 -2278.952} C_VEL
LIN {X 0,Y 573.631,Z 385.829,A -85,B 0,C 180,E1 -2281.38,E2 -2281.38} C_VEL
LIN {X 0,Y 573.782,Z 376.562,A -85,B 0,C 180,E1 -2284.294,E2 -2284.294} C_VEL
LIN {X 0,Y 573.628,Z 371.218,A -85,B 0,C 180,E1 -2286.038,E2 -2286.038} C_VEL
LIN {X 0,Y 573.267,Z 369.079,A -85,B 0,C 180,E1 -2286.812,E2 -2286.812} C_VEL
LIN {X 0,Y 573.243,Z 369.082,A -85,B 0,C 180,E1 -2289.608,E2 -2289.608} C_VEL
LIN {X 0,Y 573.245,Z 369.082,A -85,B 0,C 180,E1 -2292.642,E2 -2292.642} C_VEL
LIN {X 0,Y 573.227,Z 369.085,A -85,B 0,C 180,E1 -2295.665,E2 -2295.665} C_VEL
LIN {X 0,Y 573.235,Z 369.084,A -85,B 0,C 180,E1 -2298.543,E2 -2298.543} C_VEL
